"I_SP_T_SPANNSTELLE_3"	M 355.6	BOOL	// M-EINGANG: Spannhydraulik Taster Spannstelle 3
"I_SP_T_SPANNSTELLE_4"	M 355.7	BOOL	// M-EINGANG: Spannhydraulik Taster Spannstelle 4
"O_SP_H_SPANNSTELLE_1"	M 356.0	BOOL	// M-AUSGANG: Spannhydraulik Lampe Spannstelle 1
"O_SP_H_SPANNSTELLE_2"	M 356.1	BOOL	// M-AUSGANG: Spannhydraulik Lampe Spannstelle 2
"O_SP_H_SPANNSTELLE_3"	M 356.2	BOOL	// M-AUSGANG: Spannhydraulik Lampe Spannstelle 3
"O_SP_H_SPANNSTELLE_4"	M 356.3	BOOL	// M-AUSGANG: Spannhydraulik Lampe Spannstelle 4
"O_SP_MPL_ENTKUPPELN"	M 356.4	BOOL	// M-AUSGANG: SpannHydraulik Maschinenplatz entkuppeln
"O_SP_MPL_KUPPELN"	M 356.5	BOOL	// M-AUSGANG: SpannHydraulik Maschinenplatz kuppeln
"O_SP_RPL_AUFL_ENTSPAN"	M 356.6	BOOL	// M-AUSGANG: Ventil Luft für Auflagenkontrolle gelöst am Rüstplatz
"O_SP_RPL_AUFL_SPANNEN"	M 356.7	BOOL	// M-AUSGANG: Ventil Luft für Auflagenkontrolle gespannt am Rüstplatz
"I_AL_ANWAHL_BA1"	M 357.0	BOOL	// M-EINGANG: Freigabe Drehzahl Maximum
"I_AL_ANWAHL_BA2"	M 357.1	BOOL	// M-EINGANG: Freigabe Betriebsart 2
"I_AL_ANWAHL_BA3/4"	M 357.2	BOOL	// M-EINGANG: Freigabe Betriebsart 3/4
"I_PW_MPL_MDK_GEKUPPELT"	M 357.3	BOOL	// M-EINGANG: Medienkupplung Fraes-Drehtisch ausgefahren
"O_SP_RPL_DRUCK_AUS"	M 357.4	BOOL	// M-AUSGANG: H4-29.1 Spanndruck Rüstplatz Aus
"O_SP_RPL_ENTKUPPELN"	M 357.5	BOOL	// M-AUSGANG: SpannHydraulik Rüstplatz entkuppeln
"O_SP_RPL_KUPPELN"	M 357.6	BOOL	// M-AUSGANG: SpannHydraulik Rüstplatz kuppeln
"O_SP_RPL_BLASLUFT"	M 357.7	BOOL	// M-AUSGANG: Ventil Luft für Vorrichtung Abblasen
"O_SP_RPL_FREIGABE"	M 358.0	BOOL	// M-AUSGANG: Freigabe SpannHydraulik Rüstplatz
"O_RPL_TUER_SCHLIESSEN"	M 358.1	BOOL	// M-AUSGANG: Ventil Rüstplatztür schließen
"O_SO_WFK_KLE_KLEMMEN"	M 358.2	BOOL	// M-AUSGANG: Wiegenfräskopf Klemmung klemmen
"O_SO_WFK_KLE_LOESEN"	M 358.3	BOOL	// M-AUSGANG: Wiegenfräskopf Klemmung lösen
"O_SO_WFK_MEDIENK_REINIG"	M 358.4	BOOL	// M-AUSGANG: Wiegenfräskopf Medienkupplung abblasen/reinigen
"O_SO_WFK_PNEUMATIK_EIN"	M 358.5	BOOL	// M-AUSGANG: Wiegenfräskopf Pneumatik Ein
"O_SO_DMS_PNEUMAK_EIN"	M 358.6	BOOL	// M-AUSGANG: Drehmomentstütze Pneumatikversorgung Ein
"O_PW_MPL_MDK_ENTKUPPELN"	M 358.7	BOOL	// M-AUSGANG: Medienkupplung Fraes-Drehtisch einfahren
"I_KA_N_SPI_DURCHFLUSSW"	M 359.0	BOOL	// M-EINGANG: Durchflusswaechter Kuehlkreislauf Hauptantrieb
"I_FD_N_DURCHFL_LAGER"	M 359.1	BOOL	// M-EINGANG: Durchflusswaechter Kuehlkreislauf Lager FD-Tisch
"I_FD_NEG_DURCHFL_STATOR"	M 359.2	BOOL	// M-EINGANG: Durchflusswaechter Kuehlkreislauf Stator FD-Tisch
"I_KA_N_ACHS_DURCHFLUSSW"	M 359.3	BOOL	// M-EINGANG: Durchflusswaechter Kuehlkreislauf Vorschubantriebe
"I_AL_N_FLOW_SWITCH_3"	M 359.4	BOOL	// M-EINGANG:
"I_FD_D_TISCH_GEKLEMMT"	M 359.5	BOOL	// M-EINGANG: Diagnose Klemmung geklemmt
"I_FD_D_TISCH_GELOEST"	M 359.6	BOOL	// M-EINGANG: Diagnose Klemmung geloest
"I_FD_SCH_ZYL_SCHALTER"	M 359.7	BOOL	// M-EINGANG: Zyklenschalter Progressivverteiler
"I_FD_SCH_FUELL_OK"	M 360.0	BOOL	// M-EINGANG: Fuellstand Schmierstoffpumpe Fraes-Drehtisch
"O_WFK_aktiv"	M 360.1	BOOL	// WIKO: Betrieb mit aktivem Wiegenfräßkopf
"I_SP_SPANN_LOES"	M 360.2	BOOL	// M-EINGANG: Wahlschalter Spannhydraulik
"I_SP_AKTIV"	M 360.3	BOOL	// M-EINGANG: Freigabe Sicherheitsventil
"O_KM_FEINSTB_PUMPE"	M 360.4	BOOL	// M-AUSGANG: Foerderpumpe Feinstbereich
"O_FD_SCH_PUMPE_EIN"	M 360.5	BOOL	// M-AUSGANG: Schmierstoffpumpe ein Fraes-Drehtisch
"I_KM_WARN_KSS_TEMP"	M 361.0	BOOL	// M-EINGANG: Kuehlmittel Warnung Temperaturueberwachung
"I_KM_Leckueberw_OK"	M 361.1	BOOL	// M-EINGANG: Ueberwachung Kuehlmittel SFK
"O_PW_MPL_MDK_KUPPELN"	M 361.2	BOOL	// M-AUSGANG: Medienkupplung Fraes-Drehtisch ausfahren
"I_MessDose_BB"	M 361.3	BOOL	// M-EINGANG: Messdose Betriebsbereit
"I_WZ_MIN_SCH_Fuell_OK"	M 361.4	BOOL	// M-EINGANG: Minimalmengenschmierung Fuellstand ok
"I_AL_SCH_M26_Rueckm"	M 361.5	BOOL	// M-EINGANG: Druckueberwachung Schmierung M26 (Drehdurchführung)
"I_AL_SCH_M26_Fuellstand"	M 361.6	BOOL	// M-EINGANG: Schmierung M26 (Drehdurchführung) Füllstand
"I_WS_Grf_offen"	M 363.4	BOOL	// M-EINGANG: STA: Werkstückgreifer geöffnet
"M_FP_Quit_M206"	M 368.0	BOOL	// WIKO: Quittierung M206 Flanke positiv
"M_Quit_M206"	M 368.1	BOOL	// WIKO: Quittierung M206
"I_FD_PW_KLE_geklemmt"	M 368.2	BOOL	// M-EINGANG: Palettenklemmung Fraes-Drehtisch geklemmt
"I_FD_PW_KLE_geloest"	M 368.3	BOOL	// M-EINGANG: Palettenklemmung Fraes-Drehtisch geloest
"I_DM_Ta_Rohteil"	M 368.5	BOOL	// M-EINGANG: MSST: Taste Status Palette Rüstplatz Maschine auf Rohteil setzen
"M_write_siro_db227"	M 368.7	BOOL	// TDS: BALLUFF Ablöschen der Daten im DB227 beim Entladen
"I_DM_Ta Y-Achse plus"	M 370.0	BOOL	// M-EINGANG: MSST: Taste Y-Achse plus
"I_DM_Ta 4-Achse rechts"	M 370.1	BOOL	// M-EINGANG: MSST: Taste 4-Achse rechts
"I_DM_Ta Eilgang"	M 370.2	BOOL	// M-EINGANG: MSST: Taste Eilgang_T 29
"I_DM_Ta_5/6-Achse minus"	M 370.3	BOOL	// M-EINGANG: MSST: Taste 5/6 Achse minus_T 48
"I_DM_Ta_5/6-Achse plus"	M 370.4	BOOL	// M-EINGANG: MSST: Taste 5/6 Achse plus_T 48
"I_DM_Ta X-Achse minus"	M 370.5	BOOL	// M-EINGANG: MSST: Taste X-Achse minus_T 30
"I_DM_Ta X-Achse plus"	M 370.6	BOOL	// M-EINGANG: MSST: Taste X-Achse plus_T 28
"I_DM_Ta Z-Achse minus"	M 370.7	BOOL	// M-EINGANG: MSST: Taste Z-Achse minus_T 39
"I_DM_Ta Z-Achse plus"	M 371.0	BOOL	// M-EINGANG: MSST: Taste Z-Achse plus
"I_DM_Ta 4-Achse links"	M 371.1	BOOL	// M-EINGANG: MSST: Taste 4-Achse links_T 40
"I_DM_Ta Y-Achse minus"	M 371.2	BOOL	// M-EINGANG: MSST: Taste Y-Achse minus_T 38
"I_DM_Ta Spindel rechts"	M 371.3	BOOL	// M-EINGANG: MSST: Taste Spindel links -_T 8
"I_DM_Ta_Spindel links"	M 371.4	BOOL	// M-EINGANG: MSST: Taste Spindel rechts_T 10
"I_DM_Ta_Spindel HALT"	M 371.5	BOOL	// M-EINGANG: MSST: Taste Spindel Halt_T 9
"I_DM_Ta_Spindel_over100"	M 371.6	BOOL	// M-EINGANG: MSST: Taste Spindeloverride 100%
"I_DM_Ta_SpiOVR_erhoehen"	M 371.7	BOOL	// M-EINGANG: MSST: Taste Spindeloverride erhöhen
"I_DM_Ta_SpiOVR_reduz"	M 372.0	BOOL	// M-EINGANG: MSST: Taste Spindeloverride reduzieren
"I_DM_Ta_BHG"	M 372.1	BOOL	// M-EINGANG: MSST: Taste Bedienhandgerät
"I_DM_Ta_KMTL"	M 372.2	BOOL	// M-EINGANG: MSST: Taste Kühlmittel
"I_DM_Ta_IKZ"	M 372.3	BOOL	// M-EINGANG: MSST: Taste Innere Kühlmittel
"O_WK_NOTACHSBETRIEB"	M 373.0	BOOL	// M-AUSGANG: KometU-Achse:Notachsbetrieb
"o_uc2e1"	M 373.1	BOOL	// M-AUSGANG: KometU-Achse:Reserve PosCode 2e1
"o_uc2e2"	M 373.2	BOOL	// M-AUSGANG: KometU-Achse:Reserve PosCode 2e2
"o_uc2e3"	M 373.3	BOOL	// M-AUSGANG: KometU-Achse:Reserve PosCode 2e3
"O_WK_POSITIONIEREN"	M 373.4	BOOL	// M-AUSGANG: KometU-Achse:Reserve PosKommando
"O_WK_PARKEN"	M 373.5	BOOL	// M-AUSGANG: KometU-Achse:Reserve Parkkommando
"O_WK_ACHSBETRIEB"	M 373.6	BOOL	// M-AUSGANG: KometU-Achse:Kommando Achsbetrieb
"O_WK_QUIT_ALARM"	M 373.7	BOOL	// M-AUSGANG: KometU-Achse:Störung quittieren
"I_WK_ALARMCODE_BIT_0"	M 374.0	BOOL	// M-EINGANG: KometU-Achse:Alarmcode Bit 2e0
"I_WK_ALARMCODE_BIT_1"	M 374.1	BOOL	// M-EINGANG: KometU-Achse:Alarmcode Bit 2e1
"I_WK_ALARMCODE_BIT_2"	M 374.2	BOOL	// M-EINGANG: KometU-Achse:Alarmcode Bit 2e2
"I_WK_ALARMCODE_BIT_3"	M 374.3	BOOL	// M-EINGANG: KometU-Achse:Alarmcode Bit 2e3
"I_WK_QUIT_KOMMANDO"	M 374.4	BOOL	// M-EINGANG: KometU-Achse:Quit bei PtP, Reserve
"I_WK_NEG_ALARM"	M 374.5	BOOL	// M-EINGANG: KometU-Achse:Alarm, L-aktiv
"I_WK_NEG_WZ_AKTIV"	M 374.6	BOOL	// M-EINGANG: KometU-Achse:Werkzeug beschäftigt, L-aktiv
"I_WK_WZ_BTB"	M 374.7	BOOL	// M-EINGANG: KometU-Achse:System bereit
"I_WK_REF"	M 375.0	BOOL	// M-EINGANG: KometU-Achse:RefNocken
"I_WK_BTB"	M 375.1	BOOL	// M-EINGANG: KometU-Achse:Achse bereit
"I_WK_ENDSCHALTER_PLUS"	M 375.2	BOOL	// M-EINGANG: KometU-Achse:Vorendschalter positiv
"I_WK_ENDSCHALTER_MINUS"	M 375.3	BOOL	// M-EINGANG: KometU-Achse:Vorendschalter negativ
"m375.4"	M 375.4	BOOL	// M-EINGANG: KometU-Achse: Reserve
"m375.5"	M 375.5	BOOL	// M-EINGANG: KometU-Achse: Reserve
"m375.6"	M 375.6	BOOL	// M-EINGANG: KometU-Achse: Reserve
"m375.7"	M 375.7	BOOL	// M-EINGANG: KometU-Achse: Reserve
"m_WzwSpUAx"	M 376.0	BOOL	// KOMET U-ACHSE: Werkzeugwechsel sperren, Komet-U-Achse in Spindel.& aktiv
"m_UiSpi"	M 376.1	BOOL	// KOMET U-ACHSE: Komet-U-Achse Werkzeug in Spindel
"m_UNotBt"	M 376.2	BOOL	// KOMET U-ACHSE: Notbetrieb von Bediener gewählt
"m_LSpUAx"	M 376.3	BOOL	// KOMET U-ACHSE: Einlesesperre durch Komet U-Achse
"M_MAG_Umk_Korrektur_bei+"	M 376.4	BOOL	// MAG: Korrektur Umkehrspiel: Aktivierung bei Plusfahrt
"M_MAG_Umk_Korrektur_bei-"	M 376.5	BOOL	// MAG: Korrektur Umkehrspiel: Aktivierung bei Minusfahrt
"M_MAG_Umk_+-1_plz_ang"	M 376.6	BOOL	// MAG: Umkehrspiel: +/- 1 Platz fahren angewählt
"M_MAG_Umk_rueck_auf_plz"	M 376.7	BOOL	// MAG :Korrektur Umkehrspiel: Rückfahrt auf vorgegebenen Mag-Platz angewählt
"M_Bearb_Ende"	M 377.0	BOOL	// SINRPC: Bearbeitungsprogramm Ende
"M_Drehzahl_Sperre"	M 377.1	BOOL	// SPINDEL: Drehzahlsperre
"M_MAG_Umk_reset_korr_fp"	M 377.2	BOOL	// MAG: Korrektur Umkehrspiel: Reset Flanke Positiv
"M_MAG_Umk_kuerzesterWeg+"	M 377.3	BOOL	// MAG: Korrektur Umkehrspiel: kürzester Weg Magazinachse ins Plus
"M_MAG_Umk_kuerzesterWeg-"	M 377.4	BOOL	// MAG: Korrektur Umkehrspiel: kürzester Weg Magazinachse ins Minus
"M_MAG_Teller_Taste_dreh"	M 377.6	BOOL	// MAG: Tellermagazin Anforderung drehen über Taste
"Mx_Maschine_min_1mal_ein"	M 377.7	BOOL	// SINRPC: Maschine min einmal ein
"O_TM_TOOL_SPIPOS_LOCK"	M 378.0	BOOL	// Verriegelungszylinder ausfahren (Werkzeug verriegeln)
"I_TM_TOOL_SPIPOS_UNLKD"	M 378.1	BOOL	// eingefahren (Werkzeug entriegelt)
"I_TM_TOOL_SPIPOS_LOCKED"	M 378.2	BOOL	// ausgefahren (Werkzeug entriegelt)
"I_TM_TST_OCC"	M 378.3	BOOL	// M-EINGANG: Uebergabeplatz belegt vertikale Kette ohne TPU
"M_RS_HUBACHSE_E0_UNTEN"	M 379.0	BOOL	// PALETTENSPEICHER: Hubachse in Ebene 0 unten
"M_RS_HUBACHSE_E0_OBEN"	M 379.1	BOOL	// PALETTENSPEICHER: Hubachse in Ebene 0 oben
"M_RS_HUBACHSE_E1_UNTEN"	M 379.2	BOOL	// PALETTENSPEICHER: Hubachse in Ebene 1 unten
"M_RS_HUBACHSE_E1_OBEN"	M 379.3	BOOL	// PALETTENSPEICHER: Hubachse in Ebene 1 oben
"O_SST_SC_CL_PO_1_STATE"	M 379.4	BOOL	// MA H4-93.2 Status Auflagenkontrolle Spannstelle 1 (Meldeleuchte)
"O_SST_SC_CL_PO_2_STATE"	M 379.5	BOOL	// MA H4-93.4 Status Auflagenkontrolle Spannstelle 2 (Meldeleuchte)
"O_SST_FLUSH_ON_H"	M 379.7	BOOL	// MA B2-87.6 Ruestplatz Spuelung aktiv (Meldeleuchte)
"O_SP_HYD_RPL_LOESEDR_OK"	M 382.0	BOOL	// M-AUSGANG: Spannvorrichtung Loesedruck vorhanden
"O_SP_HYD_RPL_SPANNDR_OK"	M 382.1	BOOL	// M-AUSGANG: Spannvorrichtung Spanndruck vorhanden
"I_PW_HUB_POS1"	M 382.2	BOOL	// M-EINGANG: Palettenwechsler Hub Position 1
"I_PW_HUB_POS2"	M 382.3	BOOL	// M-EINGANG: Palettenwechsler Hub Position 2
"I_PW_HUB_POS3"	M 382.4	BOOL	// M-EINGANG: Palettenwechsler Hub Position 3
"I_SP_HYD_EIN"	M 382.5	BOOL	// M-EINGANG: Bereichsschalter Spannhydraulik Ein
"I_SP_HYD_FUEL_OK"	M 382.6	BOOL	// M-EINGANG: Spannhydraulik Ueberwachung Fuellstand
"I_SP_HYD_NEG_STOERUNG"	M 382.7	BOOL	// M-EINGANG: Spannhydraulik Motorschutzschalter ok
"I_SP_HYD_RPL_LOESEN"	M 383.0	BOOL	// M-EINGANG: Fußschalter Spannhydraulik entspannen (lösen)
"I_SP_HYD_RPL_SPANNEN"	M 383.1	BOOL	// M-EINGANG: Fußschalter Spannhydraulik spannen
"I_SP_HYD_TEMP_OK"	M 383.2	BOOL	// M-EINGANG: Spannhydraulik Temperatur ok
"M_FP_PW_Step_Forward"	M 383.3	BOOL	// PW: Schritt Vorwärts Flanke positiv
"M_FP_PW_Step_Backward"	M 383.4	BOOL	// PW: Schritt Rückwärts Flanke positiv
"M_FN_PW_Step_Forward"	M 383.5	BOOL	// PW: Schritt Vorwärts Flanke negativ
"M_FN_PW_Step_Backward"	M 383.6	BOOL	// PW: Schritt Rückwärts Flanke negativ
"O_SP_SPANNVORR_RV_EIN"	M 383.7	BOOL	// M-AUSGANG: Rückschlagventil Entspann-Leitung RPL öffnen
"Mx_APC_Disable_H67"	M 384.0	BOOL
"Mx_Pal_Fertigteil_H67"	M 384.1	BOOL
"Mx_Pal_Defekt_H67"	M 384.2	BOOL
"O_WK_KOPF_ANGEBAUT"	M 384.4	BOOL	// M-AUSGANG: U-Achse Werkzeug angebaut
"O_WK_REG_FREIGABE"	M 384.5	BOOL	// M-AUSGANG: U-Achse Reglerfreigabe
"O_SST_FIXT_CL_PO_1_CLE"	M 384.6	BOOL	// MA H4-94.2 Auflagenkontrolle Luft für Reinigung (hoher ALK-Druck)
"O_SST_SC_SENS_ACT"	M 384.7	BOOL	// MA H4-94.4 Auflagenkontrolle Luft für Messung (niedriger ALK-Druck)
"m_mag_handfunktion_-"	M 385.0	BOOL	// MAG: Handfunktion Magazinachse ins Minus drehen
"m_mag_handfunktion_+"	M 385.1	BOOL	// MAG: Handfunktion Magazinachse ins Plus drehen
"m_mag_positioniert_fp"	M 385.2	BOOL	// MAG: Handfunktion Magazinachse positioniert Flanke positiv
"M_Tast_Man_WZSp"	M 386.0	BOOL	// WZ-SPANNER:Werkzeugspanner manuell lösen
"MX_Temp_Vorw"	M 386.1	BOOL	// KM: KSA3 Vorwarnung Temporär
"M_Motor_Aus"	M 386.2	BOOL	// KM: KSA3 Motor Aus Temporär
"I_SO_WFK_ANGEDOCKT"	M 386.3	BOOL	// M-EINGANG: Wiegenfräskopf angedockt / Klemmposition erreicht
"I_SO_WFK_KLE_GEKLEMMT"	M 386.4	BOOL	// M-EINGANG: Wiegenfräskopf Klemmung geklemmt
"I_SO_WFK_KLE_GELOEST"	M 386.5	BOOL	// M-EINGANG: Wiegenfräskopf Klemmung gelöst
"I_SO_DMS_UEBERWACH_OEL"	M 386.6	BOOL	// M-EINGANG: Drehmomentstütze Ölstandsüberwachung Niveau
"I_AL_NETZAUSF_UEBERW"	M 386.7	BOOL	// ME A0-82.4 Spannungsüberwachung Netz nicht in Ordnung
"I_SP_HYD_RPL_AUS"	M 387.0	BOOL	// M-EINGANG: Ruestplatz Ventil Drucklos
"I_HYD_NEG_FILTER_RPL"	M 387.1	BOOL	// M-EINGANG: Spannhydraulik Filterverschmutzung Ruestplatz
"I_HYD_NEG_FILTER_MPL"	M 387.2	BOOL	// M-EINGANG: Spannhydraulik Filterverschmutzung Maschinenplatz
"I_ACHS_PNOZ_FRG"	M 387.3	BOOL	// M-EINGANG: Freigabe Achsen Sicherheitsschaltgeraet
"O_SP_RPL_GESPANNT"	M 387.4	BOOL	// M-AUSGANG: Spannhydraulik Ruestplatz gespannt
"O_SP_RPL_DRUCKLOS"	M 387.5	BOOL	// M-AUSGANG: Ruestplatz Ventil Drucklos
"O_SP_MPL_DRU_OK"	M 387.6	BOOL	// M-AUSGANG: Spannvorrichtung Maschine gespannt
"O_SP_RPL_SPANNEN"	M 387.7	BOOL	// Spannhydraulik Ruestplatz spannen
"O_SP_MASCHINE_ENTLADEN"	M 388.0	BOOL	// M-AUSGANG: H4-07.6 Rueckmeldung Maschine Entladen
"O_SP_SCH_EIN"	M 388.1	BOOL	// M-AUSGANG: H4-05.2 Schmierstoffpumpe Spannfutter Spannvorrichtung
"M_Vollwechsel_beendet"	M 388.2	BOOL
"M_FP_Vollwechsel_beendet"	M 388.3	BOOL
"I_AL_WARNMELD_PWR_SAG"	M 389.0	BOOL	// Spannungsüberwachung Netz
"I_SP_MASCHINE_ENTLADEN"	M 389.1	BOOL	// Maschine Entladen
"I_SP_SCH_DRUCK_OK"	M 389.2	BOOL	// Druckueberwachung Schmierung Spannfutter
"I_SP_SCH_FUELLSTAND_OK"	M 389.3	BOOL	// M-EINGANG: H4-05.5 Fuellstand Schmierung Spannfutter
"M_FP_WARN_PWR_SAG"	M 389.4	BOOL	// Positive Flanke Spannungsüberwachung Netz
"M_FP_Warnmeldung_Netz"	M 389.5	BOOL	// Impuls Spannungsüberwachung Netz
"MX_BHG_aktiv"	M 390.0	BOOL	// BHG-MPI: aktiv
"MX_FP_BHG_aktiv"	M 390.1	BOOL	// BHG-MPI: aktiv Flanke positiv
"MX_FN_BHG_aktiv"	M 390.2	BOOL	// BHG-MPI: aktiv Flanke negativ
"MX_BHG_Reset"	M 390.3	BOOL	// BHG-MPI: Reset
"MX_BHG_Anf_JOG"	M 390.4	BOOL	// BHG-MPI: Anforderung JOG
"MX_BHG_Anf_Single"	M 390.5	BOOL	// BHG-MPI: Anforderung Single Block
"MX_BHG_KM1_EinAus"	M 390.6	BOOL	// BHG-MPI: Taste Kühlmittel Ein / Aus
"MX_BHG_Handrad_aktiv"	M 390.7	BOOL	// BHG-MPI: Handrad aktiv
"MX_BHG_Taste_plus"	M 391.0	BOOL	// BHG-MPI: Taste Plus
"MX_BHG_Taste_minus"	M 391.1	BOOL	// BHG-MPI: Taste Minus
"MX_BHG_X_Vorwahl"	M 391.2	BOOL	// BHG-MPI: Vorwahl X-Achse
"MX_BHG_Y_Vorwahl"	M 391.3	BOOL	// BHG-MPI: Vorwahl Y-Achse
"MX_BHG_Z_Vorwahl"	M 391.4	BOOL	// BHG-MPI: Vorwahl Z-Achse
"MX_BHG_C_Vorwahl"	M 391.5	BOOL	// BHG-MPI: Vorwahl C-Achse
"MX_BHG_5/6_Vorwahl"	M 391.6	BOOL	// BHG-MPI: Vorwahl 5te / 6te Achse
"MX_BHG_Taste_INC1000"	M 391.7	BOOL	// BHG-MPI: Taste INC1000
"MX_BHG_Anf_INC_100"	M 392.0	BOOL	// BHG-MPI: Anforderung INC100
"MX_BHG_Anf_INC_10"	M 392.1	BOOL	// BHG-MPI: Anforderung INC10
"MX_BHG_Anf_INC_1"	M 392.2	BOOL	// BHG-MPI: Anforderung INC1
"MX_BHG_Anf_VorschHalt"	M 392.3	BOOL	// BHG-MPI: Anforderung Vorschub Halt
"MX_BHG_Anf_VorschStart"	M 392.4	BOOL	// BHG-MPI: Anforderung Vorschub Start
"MX_BHG_Anf_SpindelStart"	M 392.5	BOOL	// BHG-MPI: Anforderung Spindel Start
"MX_BHG_Anf_NC-Start"	M 392.6	BOOL	// BHG-MPI: Anforderung NC-Start
"MX_BHG_Anf_NC-Stop"	M 392.7	BOOL	// BHG-MPI: Anforderung NC-Stop
"MX_BHG_Taste_Eilgang"	M 393.0	BOOL	// BHG-MPI: Taste Eilgang
"MX_BHG_Anf_INC_1000"	M 393.1	BOOL	// BHG-MPI: Anforderung INC1000
"MX_WKS_MKS_Aend"	M 393.2	BOOL	// BHG-MPI: WKS / MKS Änderung
"MX_AX4_InPos_Fein"	M 393.3	BOOL	// BHG-MPI: Achse 4 Position erreicht mit Genauhalt fein
"MX_AX5_InPos_Fein"	M 393.4	BOOL	// BHG-MPI: Achse 5 Position erreicht mit Genauhalt fein
"MX_NC_Datueb_aktiv"	M 393.5	BOOL	// BHG-MPI: NC Datenübertragung aktiv
"MX_RD_akt_Pos_MKS"	M 393.6	BOOL	// BHG-MPI: Aktuelle Position MKS
"M_Error_WR_FC13"	M 393.7	BOOL	// BHG-MPI: Fehler Displaycontrol
"MX_RD_akt_Pos_WKS"	M 394.0	BOOL	// BHG-MPI: Aktuelle Position MKS
"M_Initialisier_Auftraege"	M 394.1	BOOL	// WIKO: Aufträge initialisieren
"I_KM_DURCHFLUSS_HD_OK"	M 394.2	BOOL	// M-EINGANG: ME C1-13.4 Durchflusswaechter Kuehlmittel 2 (M7)
"I_KM_M7_DFW_LTG_OK"	M 394.3	BOOL	// M-EINGANG: ME C1-13.7 Durchflusswaechter Leitungsueberwachung (M7)
"M_Restweg_aktiv"	M 394.4	BOOL
"M_Error_Restweg_lesen"	M 394.5	BOOL
"M_NDR_Restweg_lesen"	M 394.6	BOOL
"M_Req_Restweg_lesen"	M 394.7	BOOL
"O_SO_EXH_ON1"	M 397.0	BOOL	// Leistungssteuerung Absauganlage
"O_MT_KALIBRIER_REINIGEN"	M 397.1	BOOL	// Kalibrier Vorrichtung Messtaster abblasen
"I_KM_WARTUNG"	M 397.2	BOOL	// Filterverschmutzung Feinstbereich Warnung
"FP_SS_ROB_OFF"	M 397.3	BOOL	// Flankenmerker positiv Schlüsselschalter Robbi Aus
"FP_SS_RO"	M 397.4	BOOL	// Flankenmerker positiv Schlüsselschalter Robbi Aus
"Mx_PAldata_FASTEMS"	M 400.0	BOOL
"M_FP_Achse4_Spindel"	M 400.1	BOOL
"M_IMP_Achse4_Spindel"	M 400.2	BOOL
"M_FN_Achse4_Spindel"	M 400.3	BOOL
"M_IMP_Achse4_Achse"	M 400.4	BOOL
"M_Axpos_lesen_ready"	M 400.5	BOOL	// UT: Istwert Teil 1 gelesen
"M_184.0"	M 400.6	BOOL	// UT: NC-Datenübertragung aktiv
"M_185.6"	M 400.7	BOOL	// UT: lesen Istwert alle Achsen
"M_Axpos_read_error"	M 401.0	BOOL	// UT: Fehler Istwert lesen
"M_Req_Lesen_Ax9"	M 401.1	BOOL
"M_Error_Lesen_Ax9"	M 401.2	BOOL
"M_RDY_Lesen_Ax9"	M 401.3	BOOL
"MX_Error_RD_IstPos15"	M 401.4	BOOL
"Error_FB_SIEM_GET"	M 401.5	BOOL	// Error-Meldung Baustein FB_SIEM_GET
"NDR_FB_SIEM_GET"	M 401.6	BOOL	// NDR-Meldung Baustein FB_SIEM_GET
"MX_NDR_RD_IstPos15"	M 401.7	BOOL
"M_all_axis_pos_contr_act"	M 402.0	BOOL	// Alle aktiven Achsen befinden sich in Lageregelung
"M_PV_akt_Prg_lesen"	M 404.0	BOOL	// lesen Programmnr. aktives laufendes Programm
"M_FP_BlockSearch"	M 404.1	BOOL	// FP Satzsuchlauf aktiv
"M_M60_angewaehlt"	M 404.2	BOOL
"M_PrgLesenNCbeendet"	M 404.3	BOOL
"M_PrgLesenNC_wiederh"	M 404.4	BOOL	// Programmnummer NC lesen wiederholen bei Fehler
"M_PrgLesenNC_Fehler"	M 404.5	BOOL	// Programmnummer NC lesen Fehler gespeichert
"M_Error_Lesen_Ax16"	M 404.6	BOOL
"M_RDY_Lesen_Ax16"	M 404.7	BOOL
"M_RESET_AX16_SWN_OK"	M 405.0	BOOL
"Mx_FP_aus_Loch"	M 405.1	BOOL	// Werkzeugachse Rettung Flanke positiv
"Mx_FN_Taste"	M 405.2	BOOL	// Werkzeugachse Rettung Flanke negativ
"Mx_FN_Taste_WZ_Achse_RET"	M 405.3	BOOL	// Werkzeugachse Rettung Impuls negativ
"M_AX16_SW_NOCKEN_OK"	M 405.4	BOOL
"M_ANF_Lesen_AX16_CAM"	M 405.5	BOOL
"M_Error_Lesen_Ax16_CAM"	M 405.6	BOOL
"M_RDY_Lesen_Ax16_CAM"	M 405.7	BOOL
"M_Prog_load_unload_ok"	M 406.1	BOOL	// NC-Programm laden / entladen ok
"M_Prog_unloaded"	M 406.5	BOOL	// NC-Programm entladen
"M_Prog_loaded"	M 406.6	BOOL	// NC-Programm geladen
"I_TM_PLACE_OCCUPIED"	M 411.0	BOOL	// M-EINGANG: Magazinplatz belegt
"I_KM_DRUCK0_M7_ENABLE"	M 413.0	BOOL
"M_FN_Komet_vorhanden"	M 413.1	BOOL	// HM neg.Flanke Komet vorhanden
"Mx_SPH_DRUCK0_GESAMT_RPL"	M 413.2	BOOL	// Maschinenplatz: alle konfigurierten Spannstellen haben "Druck 0"
"Mx_SPH_DRUCK0_GESAMT_MPL"	M 413.3	BOOL	// Maschinenplatz: alle konfigurierten Spannstellen haben "Druck 0"
"I_PW_SCH_FUELLSTAND"	M 413.5	BOOL	// M-EINGANG: Schmierung Palettenwechsler Überwachung Füllstand
"I_PW_SCH_RUECKMELDUNG"	M 413.6	BOOL	// M-EINGANG: Schmierung Palettenwechsler Drucküberwachung
"O_PW_SCH_PUMPE_EIN"	M 413.7	BOOL	// M-AUSGANG: Schmierung Palettenwechsler
"I_PW_HUB_2_MITTE"	M 414.0	BOOL	// M-EINGANG: Palettenwechsler Position vor Mitte
"I_PW_HUB_2_UNTEN"	M 414.1	BOOL	// M-EINGANG: Palettenwechsler Position vor unten
"O_PW_HUB_2_HEBEN"	M 414.2	BOOL	// M-AUSGANG: Palettenwechsler Hubeinheit nach oben schnell
"O_PW_HUB_2_SENKEN"	M 414.3	BOOL	// M-AUSGANG: Palettenwechsler Hubeinheit nach unten schnell
"M_FN_KNOLL_ERROR"	M 414.4	BOOL	// KM: KNOLL Fehler Flanke negativ
"M_KNOLL_ERROR"	M 414.5	BOOL	// KM: KNOLL Fehler steht an
"M_PS_RPL_BLASLUFT_PARALL"	M 414.6	BOOL	// PALETTENSPEICHER: Blasluft Medienkupplung einschalten
"Error_FB_SIEM_GET_WZDat"	M 421.0	BOOL	// WZV: Error Greiferdaten lesen 2
"NDR_FB_SIEM_GET_WZDat"	M 421.1	BOOL	// WZV: Greiferdaten lesen fertig 2
"Req_FB_SIEM_GET_WZDat"	M 421.2	BOOL	// WZV: Request Greiferdaten lesen 2
"M_Taste_TLOAD_TOOL_LOCK"	M 421.3	BOOL
"M_FP_Zustimmtaste"	M 421.4	BOOL
"M_IM_Zustimmtaste"	M 421.5	BOOL
"M_Sperre_entr_Ladest"	M 421.6	BOOL
"M_FP_WM_Tuere_zu"	M 421.7	BOOL
"M_FP_SPH_FD_entspannen"	M 426.0	BOOL	// Impuls Spannhydraulik FD entspannen
"M_FP_Rein_Ende"	M 426.6	BOOL
"M_FN_Rett_Rein"	M 426.7	BOOL
"I_RPT_Taste_Pal_drehen"	M 427.0	BOOL	// ME xx-xx.x Taste Palette am RPL über NC-Achse drehen
"m_Req_RPAchse_drehen"	M 427.1	BOOL	// Anforderung Palette am RPL über NC-Achse drehen
"M_FP_WZ_Vorbereitet"	M 430.0	BOOL	// WZV: Quittung Bereitstellen fertig Flanke positiv
"M_FP_Reset_WZVorbereitet"	M 430.1	BOOL	// WZV: Reset Bereitstellen fertig Flanke positiv
"O_SF_Schnecke2_Maschine"	M 430.2	BOOL	// M-AUSGANG: Spaenefoerderer Schneckenantrieb 2 ein
"O_SF_Schnecke_Maschine"	M 430.3	BOOL	// M-AUSGANG: Spaenefoerderer Schneckenantrieb ein
"M_A4_loes_aktiv"	M 430.4	BOOL	// AX: Achse 4 lösen aktiv
"M_WZGr1_belegt"	M 430.5	BOOL	// WZW: Greifer 1 hat ein Werkzeug
"M_WZGr2_belegt"	M 430.6	BOOL	// WZW: Greifer 2 hat ein Werkzeug
"M_Req_GRF2_Mag"	M 430.7	BOOL	// WZW: Anforderung Greifer 2 zum Magazin
"M_FN_SPI_re.li."	M 431.0	BOOL	// MSST: Taste Spindel links / rechts Flanke negativ
"O_AL_5ACHS_KLE_LOESEN"	M 431.1	BOOL	// Klemmung loesen NC-Teilapparat
"M_WZWV_UMSPEICHERN"	M 431.2	BOOL	// WZWV: Gr2-->TPU Gr1-->Spdl / Gr1-->TPU Gr2-->Spdl Umspeichern aktivieren
"M_FP_SOKO_ERROR1"	M 431.3	BOOL	// SONDERKONSTRUKTION: SOKO Fehler 1 Flanke positiv
"M_FP_SOKO_ERROR2"	M 431.4	BOOL	// SONDERKONSTRUKTION: SOKO Fehler 2 Flanke positiv
"M_FP_KNOLL_ERROR1"	M 431.5	BOOL	// KM: KNOLL Fehler 1 Flanke positiv
"M_FP_KNOLL_ERROR2"	M 431.6	BOOL	// KM: KNOLL Fehler 2 Flanke positiv
"M_M_FKT_SPANNER_ZU_FP"	M 431.7	BOOL	// WZWV: M-Funktion Werkzeugspanner schliessen Flanke positiv
"O_AL_KABINE_ENTRIEGELN"	M 432.0	BOOL	// M-AUSGANG: Magnetverriegelung Kabinentüre entriegeln
"O_AL_PLC_BTB"	M 432.1	BOOL	// M-AUSGANG: Maschine 'Ein'  (CNC PLC Betriebsbereit)
"O_AL_Manual_Betrieb"	M 432.2	BOOL	// M-AUSGANG: Handbetrieb (Manual)
"O_Umsch_Zustimm_HR"	M 432.3	BOOL	// M-AUSGANG: Handkommandostation angewählt /Umschaltung Zustimmtasten
"O_AL_SCH_Pumpe_ein"	M 432.4	BOOL	// M-AUSGANG: Schmierung Maschine 'Ein'
"O_AL_Tempkomp_DSR"	M 432.5	BOOL	// M-AUSGANG: Temperaturkompensation rücksetzen Synchronisation Temperaturdaten
"O_AL_Tempkomp_CTS"	M 432.6	BOOL	// M-AUSGANG: Temperaturkompensation   Temperaturdaten auslesen
"M_SOKO_ERROR"	M 432.7	BOOL	// SONDERKONSTRUKTION: SOKO Fehler
"O_SK_1_Stufe_Getriebe"	M 433.0	BOOL	// M-AUSGANG: Drehzahlschaltung Hauptantrieb mit Getriebe    Drehzahl kleiner
"O_SK_2_Stufe_Getriebe"	M 433.1	BOOL	// M-AUSGANG: Drehzahlschaltung Hauptantrieb mit Getriebe    Drehzahl größer
"O_AL_Druckluft_ein"	M 433.2	BOOL	// M-AUSGANG: Pneumatik 'Ein'
"O_AL_Hydraulik_Ein"	M 433.3	BOOL	// M-AUSGANG: Hydraulik 'Ein'
"O_AL_WZ_Spanner_Loesen"	M 433.4	BOOL	// M-AUSGANG: Werkzeugspanner lösen (Autobetr)/Anwahl lösen (Handbetr)
"O_4_Klem_Bremse_Auf"	M 433.5	BOOL	// M-AUSGANG: 4.Achse Klemmung lösen
"O_5_Klem_Bremse_Auf"	M 433.6	BOOL	// M-AUSGANG: 5./11. Achse Klemmung lösen
"O_AL_Start_Sig_Renishaw"	M 433.7	BOOL	// M-AUSGANG: Messtasterfreigabe
"O_WZKegel_Blasluft"	M 434.0	BOOL	// M-AUSGANG: Messtaster Messstelle reinigen (M29) und  Werkzeugkegel ausblasen
"O_KM_M8_Ein"	M 434.1	BOOL	// M-AUSGANG: Pumpe Kühlmittel 1 'Ein' (M8)
"O_KM_M7_Ein"	M 434.2	BOOL	// M-AUSGANG: Pumpe Kühlmittel 2 'Ein' (M7)
"M_M8_Sperre_Wiko"	M 434.3	BOOL
"O_SFK_Hori_schwenken"	M 434.4	BOOL	// SCHWENKFRÄSKOPF: schwenken waagrecht (M53)
"M_M7_aktivieren_Wiko"	M 434.5	BOOL
"O_SFK_Klemmung_zu"	M 434.6	BOOL	// SCHWENKFRÄSKOPF: Klemmung klemmen
"O_SFK_Klemmung_Auf"	M 434.7	BOOL	// SCHWENKFRÄSKOPF: Klemmung lösen
"O_SPI_SCH_OEL"	M 435.0	BOOL	// M-AUSGANG: Schmierung Hauptantrieb 24.000 U/min
"O_SPI_SCH_LUFT"	M 435.1	BOOL	// M-AUSGANG: Schwenkfräskopf Druckluft Schmierung 'Ein'
"M_FR_PW_HA_SYST"	M 435.2	BOOL	// Freigabe Palettenwechsel vom Handlingsystem
"M_FN_Be_Entladen"	M 435.3	BOOL	// Abfallende Flanke: Be- Entladen aktiv
"O_Programm_Ende"	M 435.4	BOOL	// MA: Zusatzfunktion Programm Ende (M30)
"O_CNC_Fehlermeldung"	M 435.5	BOOL	// MA: Zusatzfunktion NC-Fehlermeldung steht an
"O_Funktion_M190"	M 435.6	BOOL	// M-AUSGANG: Zusatzfunktion M190
"O_PC_PAL_CAR_DOWN"	M 435.7	BOOL	// M-AUSGANG: Takttisch Palettenträger senken
"O_WM_MAG_Rechtslauf"	M 436.0	BOOL	// M-AUSGANG: Werkzeugmagazin Rechtslauf
"O_WM_MAG_Linkslauf"	M 436.1	BOOL	// M-AUSGANG: Werkzeugmagazin Linkslauf
"O_KA_STOERMELDUNG1"	M 436.2	BOOL	// M-AUSGANG: Kuehlaggregat Störmeldung Prioritaet 1
"O_PW_SPANNDRUCK_HYD_AUS"	M 436.3	BOOL	// M-AUSGANG: MA H4-03.7 Spannvorrichtung Verriegelung Palettenwechsler
"O_WZ_DATENSICHERUNG"	M 436.7	BOOL	// M-AUSGANG: Anstoss zur Datensicherung der Werkzeugdaten
"O_PW_PAL_AUF_RP_SPANNEN"	M 437.0	BOOL	// M-AUSGANG: Palette auf Rüstplatz spannen
"O_PW_PAL_AUF_RP_LOESEN"	M 437.1	BOOL	// M-AUSGANG: Palette auf Rüstplatz lösen
"O_PW_ANDOCK_SENKEN"	M 437.2	BOOL	// M-AUSGANG: Palettenwechsler Rüstplatz Andockstation senken
"O_PW_ANDOCK_HEBEN"	M 437.3	BOOL	// M-AUSGANG: Palettenwechsler Rüstplatz Andockstation heben
"O_PW_FREIGABE"	M 437.4	BOOL	// M-AUSGANG: Anforderung Freigabe Palettenwechsel
"O_WZB_Abblasen"	M 437.5	BOOL	// M-AUSGANG: Werkzeugbruchkontrolle abblasen
"O_AL_4_BA_Selbsthaltung"	M 437.7	BOOL	// M-AUSGANG: Energiefreigabe 4.Betriebsart
"O_WZB_Messung_Start"	M 438.0	BOOL	// M-AUSGANG: Werkzeugbruchüberwachung Freigabe
"O_Fenster_WZ_Mag_zu"	M 438.1	BOOL	// M-AUSGANG: Magnetverriegelung Fenster Werkzeugbestückung
"O_WM_Beladung_entr_auf"	M 438.2	BOOL	// M-AUSGANG: Freigabe Magnetverriegelung Fenster Werkzeugbestückung
"O_PW_KLE_loesen"	M 438.3	BOOL	// M-AUSGANG: Palette auf Tisch lösen
"O_PW_KLE_klemmen"	M 438.4	BOOL	// M-AUSGANG: Palette auf Tisch spannen
"O_PW_Hub_senken"	M 438.5	BOOL	// M-AUSGANG: Palettenwechsler nach unten
"O_PW_Hub_heben"	M 438.6	BOOL	// M-AUSGANG: Palettenwechsler nach oben
"O_PW_0_Grad_Drehen"	M 438.7	BOOL	// M-AUSGANG: Palettenwechsler schwenken 0 Grad Position
"O_PW_180_Grad_Drehen"	M 439.0	BOOL	// M-AUSGANG: Palettenwechsler schwenken 180 Grad Position
"O_SF_Rechtslauf"	M 439.1	BOOL	// M-AUSGANG: Rechtslauf Spaenefoerderer
"O_KM_Spruehpistole_ein"	M 439.2	BOOL	// M-AUSGANG: Pumpe Kühlmittel Spülpistole
"O_Spannhydraulik_Aus"	M 439.3	BOOL	// M-AUSGANG: Spannhydraulik entspannen
"O_AL_Blasluft_M25"	M 439.4	BOOL	// M-AUSGANG: Blasluft Kuehlung Werkzeug 'Ein'
"M_PW_Pumpe_Tischspuel"	M 439.5	BOOL	// PW: Palettenwechsler Pumpe Spülung
"M_SPI_LEITUNG_TEMP_RFG"	M 440.0	BOOL	// Spindel Leitungstemperatur: Reglerfreigabe
"M_VSP_Aktiv"	M 440.2	BOOL	// TEMPERATURKOMPENSATION: Vorsatzspindel aktiv
"O_Blasluft_Messtaster"	M 440.3	BOOL	// M-AUSGANG: Blasluft Messtaster
"M_M6_aktiv"	M 440.6	BOOL	// WZW: M6 aktiv
"M_M46_Gre_Hub_Grdst_Req"	M 440.7	BOOL	// WZW: Greifer / Hub Anforderung Grundstellung
"I_RPL_TASTE_DUSCHE_EIN"	M 441.0	BOOL	// ME G1-36.5 Bedienpult-RPL: Taste Spülung ein
"O_KM_RP_Dusche_Ventil"	M 441.1	BOOL	// MA G1-36.7 KM-Anlage Rüstplatz-Dusche Ventil Ein
"HM_PI_T_Spuelung_ein"	M 441.2	BOOL	// HM PI Rüstplatz Taste Spülung ein
"PI_RPT_T_Spuelung_ein"	M 441.3	BOOL	// PI Rüstplatz Taste Spülung ein
"O_RPL_KM_SPUELUNG_EIN"	M 441.4	BOOL	// MA xx-xx.x KM-Anlage Rüstplatz-Dusche Pumpe Ein
"M_KSA_Sammelfehler"	M 441.5	BOOL	// KSA3 Sammelfehler
"O_RPL_DUSCHE_EIN"	M 441.6	BOOL	// MA xx-xx.x KM-Anlage Rüstplatz-Dusche Meldelampe Ein
"O_Funktion_M180"	M 442.0	BOOL	// MZU: Ausgang M180
"O_Funktion_M181"	M 442.1	BOOL	// MZU: Ausgang M181
"O_Funktion_M182"	M 442.2	BOOL	// MZU: Ausgang M182
"O_Funktion_M183"	M 442.3	BOOL	// MZU: Ausgang M183
"O_Funktion_M184"	M 442.4	BOOL	// MZU: Ausgang M184
"O_Funktion_M185"	M 442.5	BOOL	// MZU: Ausgang M185
"O_Funktion_M186"	M 442.6	BOOL	// MZU: Ausgang M186
"O_Funktion_M187"	M 442.7	BOOL	// MZU: Ausgang M187
"O_Funktion_M188"	M 443.0	BOOL	// MZU: Ausgang M188
"O_Funktion_M189"	M 443.1	BOOL	// MZU: Ausgang M189
"O_KM_Pumpe_Dach"	M 443.2	BOOL	// M-AUSGANG: Spaenespuelung Dach
"O_KM_Spuelpumpe_ein"	M 443.3	BOOL	// M-AUSGANG: Spaenespuelung 'Ein'
"O_M7_Luftkuehlung"	M 443.4	BOOL	// M-AUSGANG: M7 Luftkuehlung
"O_KM_Pumpe_Dach2"	M 443.5	BOOL	// M-AUSGANG: Spaenespuelung 2 Dach
"O_WW_Rueck_MAG"	M 443.7	BOOL	// M-AUSGANG: Werkzeug-Rueckhalt ausfahren (verriegeln)
"O_WW_Hub_ZYL_in_Rein"	M 444.1	BOOL	// M-AUSGANG: Werkzeugreinigung zur Stellung Reinigen
"O_WW_Buersten_Reinigung"	M 444.3	BOOL	// M-AUSGANG: Antrieb Buerste Reinigung Werkzeugkegel
"I_ROBOT_LOCK"	M 444.4	BOOL	// ME F4-66.2 Schlüsselschalter Betriebsart Roboter gesperrt
"I_ROBOT_PROT_DOOR_CLSD"	M 444.5	BOOL	// ME F4-66.7 Werkstücklader Schutzzaun geschlossen
"O_Kab_Tuer_Entr"	M 444.7	BOOL	// M-AUSGANG: Lampe Taste Tuer Entriegeln
"O_LA_ausschwenken"	M 445.0	BOOL	// M-AUSGANG: Laser ausfahren
"O_LA_einschwenken"	M 445.1	BOOL	// M-AUSGANG: Laser einfahren
"O_LA_Sender_Ein"	M 445.2	BOOL	// M-AUSGANG: LaserFreigabe Sender
"O_LA_Empfaenger_Ein"	M 445.3	BOOL	// M-AUSGANG: Laser Freigabe Empänger
"O_LA_SCHMUTZB_AUF"	M 445.4	BOOL	// M-AUSGANG: Laser Ventil Schmutzblende
"O_LA_Sperrluft_Aus"	M 445.5	BOOL	// M-AUSGANG: Laser Ventil Sperrluft
"O_LA_ENABLE_EMPFAENGER2"	M 445.6	BOOL	// M-AUSGANG: Laser Freigabe Empänger 2
"O_WZK_Reinig_Blasluft"	M 446.0	BOOL	// M-AUSGANG: Werkzeugreinigung Blasluft
"I_GEN_OM_ID_SYNC"	M 446.1	BOOL	// M-EINGANG: Smartkey - Zeigt den START und RESTART der übertragung an (>50ms)
"I_GEN_OM_ID_CLOCK"	M 446.2	BOOL	// M-EINGANG: Smartkey - Protokoll-Taktrate. Daten können gelesen werden
"I_GEN_OM_ID_DATA_0"	M 446.3	BOOL	// M-EINGANG: Smartkey -  Daten-Spur 1
"I_GEN_OM_ID_DATA_1"	M 446.4	BOOL	// M-EINGANG: Smartkey -  Daten-Spur 2
"O_GEN_OM_ID_DATA_0"	M 446.5	BOOL	// M-AUSGANG: Smartkey -  Rückmeldung Daten-Spur 1
"O_GEN_OM_ID_DATA_1"	M 446.6	BOOL	// M-AUSGANG: Smartkey -  Rückmeldung Daten-Spur 2
"O_GEN_CNC_PGM_ACTIVE"	M 446.7	BOOL
"O_LA_WZ_ABBLASEN"	M 447.0	BOOL	// M-AUSGANG: Laser abblasen
"O_Y_Umschaltung_SPI"	M 447.1	BOOL	// M-AUSGANG: Stern Dreieck: Ausgang Stern
"O_D_Umschaltung_SPI"	M 447.2	BOOL	// M-AUSGANG: Stern Dreieck: Ausgang Dreieck
"O_PS_DREHST_BREMSE_AUF"	M 448.0	BOOL	// M-AUSGANG: Achse 9 (Palettenrundspeicher)  Bremse lüften
"O_PS_ABZIEHS_BREMSE_AUF"	M 448.1	BOOL	// M-AUSGANG: Bremse Kette 1 Palettenspeichersystem
"O_PS_RPL_BREMSE_AUF"	M 448.2	BOOL	// M-AUSGANG: Bremse Rüstplatz lüften
"O_PS_DREHST_HUB_AB"	M 448.3	BOOL	// M-AUSGANG: Ventil Dreheinheit nach unten
"O_PS_DREHST_HUB_AUF"	M 448.4	BOOL	// M-AUSGANG: Ventil Dreheinheit nach oben
"O_PS_RPL_TUER_VORN_ENTR"	M 448.5	BOOL	// M-AUSGANG: Ruestplatztuer vorn entriegeln
"O_PS_RPL_TUER_HINT_ENTR"	M 448.6	BOOL	// M-AUSGANG: Ruestplatztuer hinten entriegeln
"M_AchseNCT_loesen"	M 449.0	BOOL	// AX: NC-Teilapperat lösen
"M_AchseNCT_klemmen"	M 449.1	BOOL	// AX: NC-Teilapperat klemmen
"M_AchseNCT_Ready"	M 449.2	BOOL	// AX: NC-Teilapperat Ready mit klemmen / lösen
"M_AchseNCT_geloest"	M 449.3	BOOL	// AX: NC-Teilapperat gelöst
"M_A11_loes_aktiv"	M 449.4	BOOL	// AX: Achse 11 lösen aktiv
"I_D_PW_Tischspuelung"	M 450.0	BOOL	// M-EINGANG: Diagnose Spaenespülung Palettenwechsler
"I_D_KM_TPF_PAPIER_ENDE"	M 450.1	BOOL	// M-EINGANG: Diagnose Filterband Ende
"I_D_KM_TPF_PAPIER_WARN"	M 450.2	BOOL	// M-EINGANG: Diagnose Warnung Filterband Ende
"I_D_PW_HUB_IN_MITTE"	M 450.3	BOOL	// M-EINGANG: Palettenwechsler Diagnose Hub Pos. Mitte
"I_WW_POS_FRG_WZM"	M 450.4	BOOL	// M-EINGANG: Werkzeugwechsler Position Freigabe Werkzeugmagazin
"O_LED_Taste_Blau"	M 450.5	BOOL	// LED Taste Blau
"O_MessDose_Start"	M 450.6	BOOL	// M-AUSGANG: Laser Messdose ein
"O_WZ_MIN_SCH_MV1"	M 450.7	BOOL	// M-AUSGANG: Minimalmengen Schmierung Ventil 1 Ein
"O_AusBlasen_IKZ"	M 451.0	BOOL	// M-AUSGANG: Ausblasen IKZ Leitung
"O_AL_SCH_M26_Pumpe_ein"	M 451.1	BOOL	// M-AUSGANG: Dreh-Duchführung Ansteuerung Schmierpumpe 'Ein'
"M_SK_Sperre"	M 452.2	BOOL	// SCHWENKKOPF: Sperre
"Mx_FP_pos_Trigg_Blau"	M 453.0	BOOL	// LA:  FC_ZYLINDER Blaue Taste Flanke positiv
"Mx_FN_Blau"	M 453.1	BOOL	// LA:  FC_ZYLINDER Blaue Taste Flanke negativ
"Mx_Fp_GElb"	M 453.2	BOOL	// LA:  FC_ZYLINDER Gelbe Taste Flanke positiv
"Mx_Fn_Gelb"	M 453.3	BOOL	// LA:  FC_ZYLINDER Gelbe Taste Flanke negativ
"M_SSL_Aktiv"	M 453.7	BOOL	// WZV: NC Aktionssatz aktiv
"M_RPL_Bereich_1"	M 454.0	BOOL	// Rüstplatz Bereich 1
"M_RPL_Bereich_2"	M 454.1	BOOL	// Rüstplatz Bereich 2
"M_RPL_Bereich_3"	M 454.2	BOOL	// Rüstplatz Bereich 3
"M_RPL_Bereich_4"	M 454.3	BOOL	// Rüstplatz Bereich 4
"M_RPL_Pos_0"	M 454.4	BOOL	// Rüstplatz Position 0 Grad
"M_RPL_Pos_90"	M 454.5	BOOL	// Rüstplatz Position 90 Grad
"M_RPL_Pos_180"	M 454.6	BOOL	// Rüstplatz Position 180 Grad
"M_RPL_Pos_270"	M 454.7	BOOL	// Rüstplatz Position 270 Grad
"O_AL_ESR_AKTIV"	M 455.0	BOOL	// Rückmeldung Zyklus DM_ESR aktiv
"M_Wechsel_Prepare"	M 455.1	BOOL	// xxx
"M_T_WW_Gst_vorwaerts"	M 455.2	BOOL	// Taste Werkzeugwechsler vorwärts in Grundstellung fahren
"M_T_WW_Gst_rueckwaerts"	M 455.3	BOOL	// Taste Werkzeugwechsler rückwärts in Grundstellung fahren
"M_Tempkomp_eingefroren"	M 455.4	BOOL	// TEMPERATURKOMPENSATION: Eingefroren
"MX_IMP_W_Prep"	M 455.6	BOOL	// xxx
"MX_FP_W_Prep"	M 455.7	BOOL	// xxx
"M_out_mess_spindel"	M 456.0	BOOL	// xxx
"M_out_mess_spindel_2000"	M 456.1	BOOL	// xxx
"M_Not_aus"	M 456.3	BOOL	// MA: NOT-AUS  (*Maschine Ein)
"I_E_gerichtet"	M 456.4	BOOL	// M-EINGANG:
"I_WW_Y_inWWPos"	M 456.5	BOOL	// Y-Achse in Werkzeugwechselposition
"HM_PI_out_mess"	M 456.6	BOOL	// xxx
"PI_out_mess"	M 456.7	BOOL	// xxx
"O_AL_STILLSTAND"	M 457.0	BOOL	// M-AUSGANG: Stillstandueberwachung
"O_AL_NEG_NOTAUS"	M 457.1	BOOL	// M-AUSGANG: Not-Aus Drehzahl
"O_AL_TEST_BA"	M 457.2	BOOL	// Freigabe Drehzahl Betriebsarten
"I_WW_X_inWartePos"	M 457.4	BOOL	// X-Achse Werkzeugwechselwarteposition
"M_WW_Einzelfunktion"	M 457.5	BOOL	// xxx
"M_WW_Einzelschritt"	M 457.6	BOOL	// xxx
"I_WW_MagPlatz_frei"	M 457.7	BOOL	// M-EINGANG: Magazinplatz frei
"I_AL_5ACHS_KLE_GEKLEMMT"	M 458.0	BOOL	// M-EINGANG: Klemmung 5./11. Achse geklemmt
"O_KA2_STOERMELDUNG1"	M 458.1	BOOL	// M-AUSGANG: Kuehlaggregat 2 Störmeldung Prioritaet 1
"O_TA_KLEMMUNG_LOESEN"	M 458.2	BOOL	// M-AUSGANG: Klemmung loesen NC-Teilapparat
"O_SP_HYD_EIN"	M 458.3	BOOL	// M-AUSGANG: Spannhydraulik Pumpe ein
"O_WM_WZ_ZYL_CLAMP"	M 459.0	BOOL	// M-AUSGANG: Pneumatikzyl. Verriegelung WZ klemmen
"O_WM_WZ_ZYL_RELEASE"	M 459.1	BOOL	// M-AUSGANG: Pneumatikzylinder Verriegelung Werkzeug loesen
"I_WM_WZ_MAN_RELEASE"	M 459.2	BOOL	// M-EINGANG: Werkzeug manuell loesen
"O_WM_WZ_ZYL_RELEASE2"	M 459.3	BOOL	// M-AUSGANG: Pneumatikzylinder Verriegelung 2 Werkzeug loesen
"M_H5002_Wz_loesen"	M 459.4	BOOL	// WZW: H-Funktion 5002 Werkzeugspanner in Spindel lösen
"I_WK_SPINDEL_ABDECKUNG"	M 459.5	BOOL	// M-EINGANG: Spindel Abdeckung geschlossen
"MX_RefPkt_Achse"	M 460.0	BOOL	// AX6: (Spindel) Referenzpunkt Achse
"MX_Spdl_KorrWirksam"	M 460.1	BOOL	// AX6: (Spindel) Vorschubkorrektur wirksam setzen
"MX_Spdl_Spdl_Reset"	M 460.2	BOOL	// AX6: (Spindel) Spindel Reset
"MX_Spdl_Neu_Referenz"	M 460.3	BOOL	// AX6: (Spindel) neu Referieren
"MX_Spdl_Bei_Pos_NeuRef"	M 460.4	BOOL	// AX6: (Spindel) bei Positionieren neu Referieren
"MX_Spdl_RestwegLoeschen"	M 460.5	BOOL	// AX6: (Spindel) Restweg löschen
"I_SP_RPL_ALK_AUS"	M 460.6	BOOL	// ME H4-22.7 Schlüsselschalter Auflagekontrolle aus
"M_Req_GRF1_Mag"	M 460.7	BOOL	// WZW: Anforderung Greifer 1 zum Magazin
"MX_Spdl_PosBetr_84x5"	M 461.0	BOOL	// AX6: (Spindel) Positionierbetrieb
"MX_Spdl_DrehGrenz_83x0"	M 461.1	BOOL	// AX6: (Spindel) Drehzahlgrenze
"MX_Spdl_GewBohnre_84x3"	M 461.2	BOOL	// AX6: (Spindel) Gewindebohren aktiv
"MX_Spdl_SollBer_83x5"	M 461.3	BOOL	// AX6: (Spindel) Spindel im Sollbereich
"MX_Spdl_A_RefVerz_12x7"	M 461.4	BOOL	// AX6: (Spindel) Referenzverzögerung bei Motormessystem
"MX_Spdl_PendBetr_84x5"	M 461.5	BOOL	// AX6: (Spindel) Pendelbetrieb
"MX_Spdl_GetrUmsch_82x3"	M 461.6	BOOL	// AX6: (Spindel) Getriebeumschaltung 82x3
"MX_Spdl_E_RUCompl_94x2_"	M 461.7	BOOL	// AX6: (Spindel) Hochlauf beendet
"MX_Spdl_M3"	M 462.0	BOOL	// AX6: (Spindel) M3 (Rechtslauf) aktiv
"MX_Spdl_M4"	M 462.1	BOOL	// AX6: (Spindel) M4 (Linkslauf) aktiv
"MX_Spdl_M5"	M 462.2	BOOL	// AX6: (Spindel) M5 (Aus) aktiv
"MX_Spdl_M3_M4"	M 462.3	BOOL	// AX6: (Spindel) M3 oder M4 oder Fahrbefehl aktiv
"MX_Spdl_IMP_M3"	M 462.4	BOOL	// AX6: (Spindel) M3 (Rechtslauf) aktiv Impuls
"MX_Spdl_IMP_M4"	M 462.5	BOOL	// AX6: (Spindel) M4 (Linkslauf) aktiv Impuls
"MX_Spdl_IMP_M5"	M 462.6	BOOL	// AX6: (Spindel) M5 (Aus) aktiv Impuls
"MX_Spdl_IMP_M3_M4"	M 462.7	BOOL	// AX6: (Spindel) M3 oder M4 Impuls
"MX_Spdl_Reset_M3_4"	M 463.0	BOOL	// AX6: (Spindel) Reset M3 oder M4
"MX_Spdl_M3_Aktiv"	M 463.1	BOOL	// AX6: (Spindel) M3 (Rechtslauf) aktiv
"MX_Spdl_M4_Aktiv"	M 463.2	BOOL	// AX6: (Spindel) M3 (Linksslauf) aktiv
"MX_Spdl_FP_M4"	M 463.3	BOOL	// AX6: (Spindel) M4 (Linksslauf) aktiv Flanke positiv
"MX_Spdl_FP_M3"	M 463.4	BOOL	// AX6: (Spindel) M3 (Rechtslauf) aktiv Flanke positiv
"MX_Spdl_FP_M5"	M 463.5	BOOL	// AX6: (Spindel) M5 (Aus) aktiv Flanke positiv
"MX_Spdl_Hochlauf"	M 463.6	BOOL	// Spdl: Hochlauf nach Vorschub Halt
"MX_Spdl_Message_94x7"	M 463.7	BOOL	// AX6: (Spindel) Variable Meldefunktion
"MX_2GETR_VorFreig"	M 474.0	BOOL	// Getriebe: VorschubFreigabe
"MX_2Getr_AnfStufe"	M 474.1	BOOL	// Getriebe: Anforderung Stufe
"MX_2Getr_Aktiv"	M 474.2	BOOL	// Getriebe: Schalten Aktiv
"MX_2Getr_FP_Schalten"	M 474.3	BOOL	// Getriebe: Flanke Schalten
"MX_2Getr_FehlAus"	M 474.4	BOOL	// Getriebe: Fehler ausgegeben
"MX_Hawe_Ventil_0Sig"	M 474.5	BOOL	// Hawe Ventile Reitstock/Greifer 0Signal
"M_WZVS_M77_aktiviert"	M 474.6	BOOL	// WZVS mit M77 aktiviert
"Error_FC_SIEM_PLC_NCK"	M 474.7	BOOL	// Error-Meldung Baustein FC_SIEM_PLC_NCK
"I_MT_KAL_KLAPPE_ZU"	M 475.0	BOOL	// ME G5-14.3 Klappe Kalibriervorrichtung geschlossen
"I_MT_KALIBRIER_AUSG"	M 475.1	BOOL	// ME G5-14.5 Kalibrier Vorrichtung Messtaster ausgefahren
"I_MT_KALIBRIER_EING"	M 475.2	BOOL	// ME G5-14.6 Kalibrier Vorrichtung Messtaster eingefahren
"O_MT_KALIBRIER_AUSF"	M 475.3	BOOL	// MA G5-13.2 Kalibrier Vorrichtung Messtaster ausfahren
"O_MT_KALIBRIER_EINF"	M 475.4	BOOL	// MA G5-13.4 Kalibrier Vorrichtung Messtaster einfahren
"Mx_KSA_war_Aktiv"	M 475.5	BOOL	// Rückmeldung das ein M7,M8 angestanden hat
"Mx_Rauchnebel_fertig"	M 475.6	BOOL	// Rückmeldung Rauchnebelabscheider ist fertig
"mx_fn_rauchnebel"	M 475.7	BOOL	// Impuls für Rauchnebelabscheider
"M_SP_Vorschm_Req"	M 476.0	BOOL	// Spindelschmierung: Anforderung Vorschmierung
"M_WW_Bild_freifahren"	M 476.1	BOOL
"I_WW_MagTasche_auf"	M 476.2	BOOL	// M-EINGANG:
"I_WW_MagTasche_zu"	M 476.3	BOOL	// M-EINGANG:
"M_Vorschm_Imp_Ende"	M 476.4	BOOL
"M_Schmier_Imp_Ende"	M 476.5	BOOL
"M_SP_Nachschm_Req"	M 476.6	BOOL
"MX_IKZ_WZ_war_aktiv"	M 476.7	BOOL
"m_pw_schmier_stoe_dr_gsp"	M 477.0	BOOL	// Schmierung Palettenwechsler: Störung Druckaufbau gespeichert
"m_pw_start_aktiv_fp"	M 477.1	BOOL	// Palettenwechsler Start aktiv positive Flanke
"m_pw_Hub_Pos4_fn"	M 477.2	BOOL	// Position PW-Hub heben schnell
"m_pw_Hub_Pos4_fp"	M 477.3	BOOL	// Position PW-Hub senken schnell
"m_PWFG_unterdruecken"	M 477.4	BOOL	// Wegen "Schutzzaun-Funktionen" PW-Freigabe unterdruecken
"HM_PI_PWFG_unterdruecken"	M 477.5	BOOL	// HM PI Auslöser PW-Freigabe unterdrücken
"MX_FN_WZW_NC_Aktiv"	M 477.7	BOOL	// Flanke Negativ WZW NC aktiv
"IX_TLB_BIT_0"	M 500.0	BOOL	// M-EINGANG: WZB Binärcodiert
"IX_TLB_BIT_1"	M 500.1	BOOL	// M-EINGANG: WZB Binärcodiert
"IX_TLB_BIT_2"	M 500.2	BOOL	// M-EINGANG: WZB Binärcodiert
"IX_TLB_BIT_3"	M 500.3	BOOL	// M-EINGANG: WZB Binärcodiert
"IX_TLB_MEASURING_END"	M 500.4	BOOL	// M-EINGANG: WZB Messung Ende
"IX_TLB_HOME_POS"	M 500.5	BOOL	// M-EINGANG: WZB Parkstellung
"MX_Mag_Trigg4"	M 501.4	BOOL	// MAG: Trigger 4  (FC_MAG_HAUPT_ZH)
"MX_Mag_Trigg5"	M 501.5	BOOL	// MAG: Trigger 5  (FC_MAG_HAUPT_ZH)
"O_WM_Freigabe_re_li"	M 501.6	BOOL	// M-AUSGANG: Freigabe Werkzeugmagazin
"M_SK_Sicherpos"	M 503.0	BOOL
"M_AUTO_MAG_TOOL_RIEG_LOC"	M 504.0	BOOL
"M_AUTO_MAG_TOOL_RIEG_UNL"	M 504.1	BOOL
"M_K2_Programm_Aktiv"	M 504.2	BOOL
"M_K2_Vorschub_Halt"	M 504.3	BOOL
"I_TP_CALIBRATION_MOV_OU"	M 506.0	BOOL	// Messeinrichtung Messtaster ausgefahren
"I_TP_CALIBRATION_MOV_IN"	M 506.1	BOOL	// Messeinrichtung Messtaster eingefahren
"I_TP_CAL_FLAP_CLSD"	M 506.2	BOOL	// Klappe Messeinrichtung Geschlossen
"O_TP_CALIBRATION_EXTEND"	M 506.3	BOOL	// Messeinrichtung Messtaster ausfahren
"O_TP_CALIBRATION_RUN-IN"	M 506.4	BOOL	// Messeinrichtung Messtaster einfahren
"O_TP_CALIBRATION_CLEAN"	M 506.5	BOOL	// Messeinrichtung Messtaster abblasen
"MX_Ready_TM_TRANS"	M 507.0	BOOL
"M_H5000_H5004_WW_Start"	M 507.1	BOOL
"M_11Ax_plus"	M 510.0	BOOL
"M_11Ax_minus"	M 510.1	BOOL
"m_rqwwgf"	M 514.0	BOOL	// Autom.Grundstlg.fahren:Schritt Werkzeugwechsler Gf.
"m_rqpwgf"	M 514.1	BOOL	// Autom.Grundstlg.fahren:Schritt Palettenwechsler Gf.
"m_rqlagf"	M 514.2	BOOL	// Autom.Grundstlg.fahren: Schritt Laser Gf.
"M_LASER_IN_GRDST"	M 514.7	BOOL	// Laser Werkzeugvermessung in Grundstellung
"M_SO_DMS_PNEUMAK_EIN"	M 515.0	BOOL
"m_clrAl"	M 515.7	BOOL	// autom.Grundstlg.fahren:Reset Fehler/Meldungen
"M_FP_HubZyl_Start"	M 520.0	BOOL
"M_Fehl_WZB_Grdst"	M 520.1	BOOL
"M_Fehl_WZB_Grdst2"	M 520.2	BOOL
"M_FP_SPL_OK"	M 520.3	BOOL
"mx_fn_achs11"	M 520.7	BOOL
"I_KM_SF_KRATZ_NIV_MAX"	M 521.0	BOOL	// M-EINGANG: Max. Niveau-Überwachung  Kratzerförderer
"I_D_KM_SF_KRATZ_NIV_MAX"	M 521.1	BOOL	// M-EINGANG: Diagnose Max. Niveau-Überwachung  Kratzerförderer
"I_KM_SF_PUMPE_EIN"	M 521.2	BOOL	// M-EINGANG: Niveaukontrolle Schmutztank Hebepumpe „Ein“
"I_D_KM_SF_NEG_PUMPE_EIN"	M 521.3	BOOL	// M-EINGANG: Diagnose Niveau Schmutztank Hebepumpe „Ein“
"I_KM_SF_PUMPE_AUS"	M 521.4	BOOL	// M-EINGANG: Niveaukontrolle Schmutztank Hebepumpe „Aus“
"I_D_KM_SF_NEG_PUMPE_AUS"	M 521.5	BOOL	// M-EINGANG: Diagnose Niveau Schmutztank Hebepumpe „Aus“
"I_KM_SF_TANK_NIV_MAX"	M 521.6	BOOL	// M-EINGANG: Maximale Niveaukontrolle Schmutztank
"I_D_KM_SF_NEG_TANK_MAX"	M 521.7	BOOL	// M-EINGANG: Diagnose Maximale Niveaukontrolle Schmutztank
"I_TT_ausgeschwenkt"	M 522.0	BOOL	// M-EINGANG: Messtaster Tisch TS27R ausgeschwenkt
"I_TT_eingeschwenkt"	M 522.1	BOOL	// M-EINGANG: Messtaster Tisch TS27R eingeschwenkt
"O_KM_SF_KRATZER_EIN_V"	M 522.2	BOOL	// M-AUSGANG: Antrieb Kratzerförderer „Ein“
"O_KM_SF_HEBEPUMPE_EIN"	M 522.3	BOOL	// M-AUSGANG: Hebepumpe Schmutztank „Ein“
"O_AL_Messsignal_Umsch"	M 522.4	BOOL	// M-AUSGANG: Umschaltung Messsignale MesstasterTS27 / Laser
"O_TT_ausschwenken"	M 522.5	BOOL	// M-AUSGANG: Messtaster Tisch TS27R ausschwenken
"O_TT_einschwenken"	M 522.6	BOOL	// M-AUSGANG: Messtaster Tisch TS27R einschwenken
"O_TM_TPU_GET_TOOL"	M 523.0	BOOL	// M-AUSGANG: Transporteinheit auf Werkzeugkegel fahren
"I_TM_TPU_GET_TOOL"	M 523.1	BOOL	// M-EINGANG: Transporteinheit ist auf Werkzeugkegel gefahren
"O_TM_TPU_RELEASE_TOOL"	M 523.2	BOOL	// M-AUSGANG: Transporteinheit vom Werkzeugkegel wegfahren
"I_TM_TPU_RELEASE_TOOL"	M 523.3	BOOL	// M-EINGANG: Transporteinheit ist vom Werkzeugkegel weggefahren
"O_TM_TPU_TRANSFERPOS"	M 523.4	BOOL	// M-AUSGANG: Transporteinheit zu Übergabeposition fahren
"I_TM_TPU_TRANSFERPOS"	M 523.5	BOOL	// M-EINGANG: Transporteinheit ist zur Übergabeposition gefahren
"O_TM_TPU_MAGAZINPOS"	M 523.6	BOOL	// M-AUSGANG: Transporteinheit zur Magazinposition fahren
"I_TM_TPU_MAGAZINPOS"	M 523.7	BOOL	// M-EINGANG: Transporteinheit ist zur Magazinposition gefahren
"O_TM_MAG_TOOL_UNLOCK"	M 524.0	BOOL	// M-AUSGANG: Werkzeug an Magazinposition entriegeln
"I_TM_MAG_TOOL_UNLOCK"	M 524.1	BOOL	// M-EINGANG: Werkzeug an Magazinposition ist entriegelt (Zylinder)
"O_TM_MAG_TOOL_LOCK"	M 524.2	BOOL	// M-AUSGANG: Werkzeug an Magazinposition verriegeln
"I_TM_MAG_TOOL_LOCK"	M 524.3	BOOL	// M-EINGANG: Werkzeug an Magazinposition ist verriegelt (Zylinder)
"O_TM_TPU_AIR_CLEANING"	M 524.4	BOOL	// M-AUSGANG: Druckluftreinigung der Transporteinheit einschalten
"O_TM_TLOAD_TOOL_UNLOCK"	M 524.5	BOOL	// M-AUSGANG: Werkzeug am Rüstplatz entriegeln
"I_TM_TLOAD_TOOL_UNLOCK"	M 524.6	BOOL	// M-EINGANG: Werkzeug am Rüstplatz ist entriegelt (Zylinder)
"O_TM_TLOAD_TOOL_LOCK"	M 524.7	BOOL	// M-AUSGANG: Werkzeug am Rüstplatz verriegeln
"I_TM_TLOAD_TOOL_LOCK"	M 525.0	BOOL	// M-EINGANG: Werkzeug am Rüstplatz ist verriegelt (Zylinder)
"I_TM_TLOAD_PIN_LOCK"	M 525.1	BOOL	// M-EINGANG: Verriegelungspin Rüstplatz verriegelt (Kontrollschalter)
"I_TM_MAG_PIN_LOCK"	M 525.2	BOOL	// M-EINGANG: Verriegelungspin Magazinposition verriegelt (Kontrollschalter)
"M_SPI_belegt"	M 525.3	BOOL	// WZW: Werkzeug in der Spindel
"M_CU_Aktiv"	M 525.4	BOOL
"M_TPU_belegt"	M 525.5	BOOL
"M_Frg_WZ_vorbereiten"	M 525.6	BOOL
"M_Frg_WZ_ablegen"	M 525.7	BOOL
"M_WW_X_imArbeitsraum"	M 526.0	BOOL	// X-Achse im Arbeitsraum (bei Kettenmagazin)
"M_WZW_Transfer_Stellung"	M 526.1	BOOL
"NDR_WZDat_Lesen_2"	M 526.2	BOOL
"ERROR_WZDat_Lesen_2"	M 526.3	BOOL
"REQ_WZDat_Lesen_2"	M 526.4	BOOL
"I_TM_TLOAD_ACK_TOOL_IN"	M 526.5	BOOL
"I_TM_TLOAD_ACK_TOOL_OUT"	M 526.6	BOOL
"O_TM_TLOAD_TIN_H"	M 526.7	BOOL
"O_TM_TLOAD_TOUT_H"	M 527.0	BOOL
"M_Umsp_Wst_TPU"	M 527.1	BOOL
"M_Umsp_TPU_WST"	M 527.2	BOOL
"HM_PI_TM_VERW_1"	M 527.3	BOOL
"M_Umsp_Gr2_TPU"	M 527.4	BOOL
"HM_PI_TM_VERW_2"	M 527.5	BOOL
"M_Umsp_Gr1_TPU"	M 527.6	BOOL
"I_WW_X_inWWPos"	M 527.7	BOOL
"HM_PI_TM_VERW_3"	M 528.0	BOOL
"M_Umsp_TPU_Gr2"	M 528.1	BOOL
"HM_PI_TM_VERW_4"	M 528.2	BOOL
"M_AUTO_TPU_GET_TOOL"	M 528.3	BOOL
"M_AUTO_TPU_RELEASE_TOOL"	M 528.4	BOOL
"M_AUTO_TPU_MAGAZINPOS"	M 528.5	BOOL
"M_AUTO_TPU_TRANSFERPOS"	M 528.6	BOOL
"M_AUTO_MAG_TOOL_UNLOCK"	M 528.7	BOOL
"M_AUTO_MAG_TOOL_LOCK"	M 529.0	BOOL
"M_WZW_Fehler_Uebergabepl"	M 529.1	BOOL
"M_Schrittkette_Stop"	M 529.2	BOOL	// WZW: Schrittkette gestoppt durch Fehler
"M_WZW_SKZ_VOR"	M 529.3	BOOL
"M_WZW_FRG_SKZ_VOR"	M 529.4	BOOL
"M_WZW_SKZ_ZURUECK"	M 529.5	BOOL
"M_WZW_FRG_SKZ_ZURUECK"	M 529.6	BOOL
"M_WZW_GRDST_FAHRT_AKTIV"	M 529.7	BOOL
"M_FP_Greifer_drehen"	M 530.0	BOOL
"M_FN_Greifer_drehen"	M 530.1	BOOL
"M_PF_RF_X_Arbeitsraum"	M 530.2	BOOL
"M_PF_RF_X_WW_Pos"	M 530.3	BOOL
"M_PF_RF_Y_WW_Pos"	M 530.4	BOOL
"M_PF_RF_SPI_WW_Pos"	M 530.5	BOOL
"M_PF_RF_WW_180"	M 530.6	BOOL
"M_PF_RF_WW_360"	M 530.7	BOOL
"m_pWZWAsupAbbrechen"	M 531.0	BOOL	// WZW: Reset auslösen bei Abbruch Asup durch loslassen der Rettungs-Taste HM
"m_WZWAsupAbbrechen"	M 531.1	BOOL	// WZW: Reset auslösen bei Abbruch Asup durch loslassen der Rettungs-Taste
"M_FP_SKZ_VOR"	M 531.2	BOOL
"M_FP_SKZ_SAVE_RESET"	M 531.3	BOOL
"M_Frg_WW_Endstellung"	M 531.4	BOOL
"M_WW_Sperre_Wechsler"	M 531.5	BOOL
"Mx_Klappe_WZW_zu"	M 531.6	BOOL
"M_Greifer_rechts"	M 531.7	BOOL
"M_Greifer_links"	M 532.0	BOOL
"M_Grf1_0_Grad"	M 532.1	BOOL
"M_Grf1_180_Grad"	M 532.2	BOOL
"M_FN_Greifer drehen"	M 532.3	BOOL
"M_FP_SKZ_ZURUECK"	M 532.4	BOOL
"M_FP_Grf1_0_Grad"	M 532.5	BOOL
"M_FP_Grf1_180_Grad"	M 532.6	BOOL
"M_AUTO_TLOAD_TOOL_LOCK"	M 532.7	BOOL
"M_AUTO_TLOAD_TOOL_UNLOCK"	M 533.0	BOOL
"M_SperreMag_Wz_einlegen"	M 533.1	BOOL
"M_VSP_Mag_Vertikalkette"	M 533.2	BOOL
"I_DM_Ta_NC-Start"	M 533.3	BOOL
"I_WWT_offen"	M 533.4	BOOL
"I_WMT_verriegelt"	M 533.5	BOOL
"I_TM_TLOAD_TOOL_INSERT"	M 533.6	BOOL	// M-EINGANG: Positionsüberwachung Werkzeug Rüstplatz
"M_MTH_READY_SOKO"	M 534.0	BOOL
"I_PS_RPL_DREHZAHL_BIT_1"	M 534.4	BOOL	// Drehzahl Ruestplatz binaer codiert 2\20
"I_PS_RPL_DREHZAHL_BIT_2"	M 534.5	BOOL	// Drehzahl Ruestplatz binaer codiert 2\21
"I_PS_RPL_DREHZAHL_BIT_3"	M 534.6	BOOL	// Drehzahl Ruestplatz binaer codiert 2\22
"I_PS_RPL_DREHZAHL_BIT_4"	M 534.7	BOOL	// Drehzahl Ruestplatz binaer codiert 2\23
"m_request_qeifer_WZ_Gr"	M 535.0	BOOL	// Request lesen Greifer OEM Daten
"M_WZ_Wasch_schnell"	M 535.1	BOOL	// Wz Waschen 1 Sekunde aus Wz Verwaltung
"M_WZ_Wasch_abgewaehlt"	M 535.2	BOOL	// Waschen von WZ verwaltung abgewählt
"m_FLM_request_read"	M 535.3	BOOL	// FLM fuer Lesen Greifer OEM Daten
"m_VSH_SP_GETRIEBE"	M 535.4	BOOL	// Vorschubhalt von Ueberwachung Getriebeumschaltung Spindel
"O_WK_MAG_AUSFAHREN"	M 535.5	BOOL	// Werkzeugtraeger ausfahren
"O_WK_MAG_EINFAHREN"	M 535.6	BOOL	// Werkzeugtraeger einfahren
"I_WK_GRUNDSTELL"	M 535.7	BOOL	// Werkzeugtraeger Grundstellung
"I_WK_WECH_POS"	M 536.0	BOOL	// Werkzeugtraeger Wechselposition
"O_WK_ZYL_2_AUSF"	M 536.1	BOOL	// Werkzeugtraeger Zylinder 2 ausfahren
"O_WK_ZYL_2_EINFAHREN"	M 536.2	BOOL	// Werkzeugtraeger Zylinder 2 einfahren
"I_WK_ZYL_2_GST"	M 536.3	BOOL	// Werkzeugtraeger Zylinder 2 Grundstellung
"I_WK_ZYL_2_WE_POS"	M 536.4	BOOL	// Werkzeugtraeger Zylinder 2 Wechselposition
"O_WK_KLAPPE_AUF"	M 536.5	BOOL	// Werkzeugklappe oeffnen
"O_WK_KLAPPE_ZU"	M 536.6	BOOL	// Werkzeugklappe schliessen
"I_WK_KLAPPE_AUF"	M 536.7	BOOL	// Werkzeugklappe geoeffnet
"I_WK_KLAPPE_ZU"	M 537.0	BOOL	// Werkzeugklappe geschlossen
"I_WK_WZ_1_VORHANDEN"	M 537.1	BOOL	// Winkelfraeskopf 1 vorhanden
"I_WK_WZ_2_VORHANDEN"	M 537.2	BOOL	// Winkelfraeskopf 2 vorhanden
"M_VSH_GetrUeberw_aktiv"	M 537.7	BOOL	// Vorschub-Halt Überwachung Getriebeumschaltung aktiv (gespeichert)
"M_WK_Auto_Klappe_oeffnen"	M 538.0	BOOL
"M_WK_Auto_Pos1_AST"	M 538.1	BOOL
"M_WK_Auto_Pos2_AST"	M 538.2	BOOL
"M_WK_Auto_Grdst"	M 538.3	BOOL
"M_WK_Auto_Zyl2_Grdst"	M 538.4	BOOL
"M_WK_Auto_Klappe_schlies"	M 538.5	BOOL
"M_WIKO_Asup_abbrechen"	M 538.6	BOOL	// WIKO: Reset auslösen bei Abbruch Asup durch loslassen der Rettungs-Taste
"M_PW_Asup_abbrechen"	M 538.7	BOOL	// PW: Reset auslösen bei Abbruch Asup durch loslassen der Rettungs-Taste
"M_SBH_AKTIV_ARBEITSRAUM"	M 539.0	BOOL	// SAFETY: SBH aktiv -> Freigabe Arbeitsraumtüre entriegeln
"M_SBH_AKTIV_RÜSTPLATZ"	M 539.1	BOOL	// SAFETY: SBH aktiv -> Freigabe Rüstplatztüre Palettenwechsler entriegeln
"M_SBH_AKTIV_MAGAZIN"	M 539.2	BOOL	// SAFETY: SBH aktiv -> Freigabe Magazintüre entriegeln
"M_SBH_AKTIV_RPL_PS"	M 539.3	BOOL	// SAFETY: SBH aktiv -> Freigabe Rüstplatztüre Palettenspeicher entriegeln
"M_SBH_ANF_ARBEITSRAUM"	M 539.4	BOOL	// SAFETY: SBH Anforderung Arbeitsraum
"M_SBH_ANF_RÜSTPLATZ"	M 539.5	BOOL	// SAFETY: SBH Anforderung Palettenwechsler
"M_SBH_ANF_MAGAZIN"	M 539.6	BOOL	// SAFETY: SBH Anforderung Magazin
"M_SBH_ANF_RPL_PS"	M 539.7	BOOL	// SAFETY: SBH Anforderung  Palettenspeicher
"M_Umsp_TPU_Gr1"	M 540.0	BOOL
"M_FN_RP_Palette_weg"	M 540.1	BOOL
"M_FN_RP_Pal_auf_0"	M 540.2	BOOL
"M_Kegelrein_VM_aktiv"	M 540.3	BOOL
"M_Anwahl_WZW_Maske"	M 540.7	BOOL	// Anwahl für Maske Schneller Werkzeugwechsel
"I_TM_TOOL_CYL_LOCKED"	M 541.0	BOOL
"I_TM_TOOL_CYL_UNLOCKED"	M 541.1	BOOL
"M_AUTO_TLOAD_CYL_LOCK"	M 541.2	BOOL
"M_AUTO_TLOAD_CYL_UNLOCK"	M 541.3	BOOL
"O_TM_TOOL_CYL_LOCK"	M 541.4	BOOL
"M_FP_Auto_TLoad_Tool_Loc"	M 541.5	BOOL
"M_FN_Te_Pin_Ruest_Lock"	M 541.6	BOOL
"M_FP_TLOAD_TOOL_LOCK"	M 541.7	BOOL
"m_oem_freigabe_bew_nr"	M 549.0	BOOL	// OEM: Freigabe OEM Bewegungsnummer (Taste Blau/Gelb aktiv)
"m_oem_reset_frg_bew_nr"	M 549.1	BOOL	// OEM: Reset Freigabe OEM Bewegungsnummer Flanke Positiv
"M_FP_Achse14_steht"	M 549.2	BOOL
"M_FP_Achse_WZGR_Pos_lese"	M 549.3	BOOL
"M_FP_Einlesesperre"	M 549.7	BOOL
"m_hmi_pro_taste_plus"	M 550.0	BOOL	// HMI-PRO: Taste plus
"m_hmi_pro_taste_minus"	M 550.1	BOOL	// HMI-PRO: Taste minus
"m_550.2"	M 550.2	BOOL	// HMI-PRO:
"m_550.3"	M 550.3	BOOL	// HMI-PRO:
"m_550.4"	M 550.4	BOOL	// HMI-PRO:
"m_550.5"	M 550.5	BOOL	// HMI-PRO:
"m_550.6"	M 550.6	BOOL	// HMI-PRO:
"m_550.7"	M 550.7	BOOL	// HMI-PRO:
"m_hmi_pro_m551.0"	M 551.0	BOOL	// HMI-PRO: Bild Einschaltbedingungen -
"m_hmi_pro_m551.1"	M 551.1	BOOL	// HMI-PRO: Bild Einschaltbedingungen -
"m_hmi_pro_HYD_einschalt"	M 551.2	BOOL	// HMI-PRO: Bild Einschaltbedingungen -  Hydraulik EIN
"m_hmi_pro_HYD_ausschalt"	M 551.3	BOOL	// HMI-PRO: Bild Einschaltbedingungen -  Hydraulik AUS
"m_hmi_pro_PNEU_einschalt"	M 551.4	BOOL	// HMI-PRO: Bild Einschaltbedingungen -  Pneumatik EIN
"m_hmi_pro_PNEU_ausschalt"	M 551.5	BOOL	// HMI-PRO: Bild Einschaltbedingungen -  Pneumatik AUS
"m_hmi_pro_KMTL_einschalt"	M 551.6	BOOL	// HMI-PRO: Bild Einschaltbedingungen -  Kühlmitelanlage EIN
"m_hmi_pro_KMTL_ausschalt"	M 551.7	BOOL	// HMI-PRO: Bild Einschaltbedingungen -  Kühlmitelanlage AUS
"m_552.0"	M 552.0	BOOL	// HMI-PRO:
"m_552.1"	M 552.1	BOOL	// HMI-PRO:
"m_552.2"	M 552.2	BOOL	// HMI-PRO:
"m_552.3"	M 552.3	BOOL	// HMI-PRO:
"m_552.4"	M 552.4	BOOL	// HMI-PRO:
"m_552.5"	M 552.5	BOOL	// HMI-PRO:
"m_552.6"	M 552.6	BOOL	// HMI-PRO:
"m_552.7"	M 552.7	BOOL	// HMI-PRO:
"m_hmi_pro_HYD_ein_gesp"	M 553.0	BOOL	// HMI-PRO: Bild Einschaltbedingungen - Hydraulik EIN gespeichert
"m_hmi_pro_PNEU_ein_gesp"	M 553.1	BOOL	// HMI-PRO: Bild Einschaltbedingungen - Pneumatik EIN gespeichert
"m_553.2"	M 553.2	BOOL	// HMI-PRO:
"m_553.3"	M 553.3	BOOL	// HMI-PRO:
"m_553.4"	M 553.4	BOOL	// HMI-PRO:
"m_553.5"	M 553.5	BOOL	// HMI-PRO:
"m_553.6"	M 553.6	BOOL	// HMI-PRO:
"m_553.7"	M 553.7	BOOL	// HMI-PRO:
"m_hmi_pro_zeile_mb554.0"	M 554.0	BOOL	// HMI-PRO: Byte Einrichtzeilennummer
"m_hmi_pro_zeile_mb554.1"	M 554.1	BOOL	// HMI-PRO: Byte Einrichtzeilennummer
"m_hmi_pro_zeile_mb554.2"	M 554.2	BOOL	// HMI-PRO: Byte Einrichtzeilennummer
"m_hmi_pro_zeile_mb554.3"	M 554.3	BOOL	// HMI-PRO: Byte Einrichtzeilennummer
"m_hmi_pro_zeile_mb554.4"	M 554.4	BOOL	// HMI-PRO: Byte Einrichtzeilennummer
"m_hmi_pro_zeile_mb554.5"	M 554.5	BOOL	// HMI-PRO: Byte Einrichtzeilennummer
"m_hmi_pro_zeile_mb554.6"	M 554.6	BOOL	// HMI-PRO: Byte Einrichtzeilennummer
"m_hmi_pro_zeile_mb554.7"	M 554.7	BOOL	// HMI-PRO: Byte Einrichtzeilennummer
"m_hmi_pro_m555.0"	M 555.0	BOOL	// HMI-PRO: Taktart -
"m_hmi_pro_leerfahren_akt"	M 555.1	BOOL	// HMI-PRO: Taktart - Leerfahren aktiv
"m_hmi_pro_warmfahren_akt"	M 555.2	BOOL	// HMI-PRO: Taktart - Warmfahren aktiv
"m_hmi_pro_fahren_oW_akt"	M 555.3	BOOL	// HMI-PRO: Taktart - Fahren ohne Werkstück aktiv
"m_555.4"	M 555.4	BOOL	// HMI-PRO: Taktart -
"m_555.5"	M 555.5	BOOL	// HMI-PRO: Taktart -
"m_555.6"	M 555.6	BOOL	// HMI-PRO: Taktart -
"m_555.7"	M 555.7	BOOL	// HMI-PRO: Taktart -
"m_556.0"	M 556.0	BOOL	// HMI-PRO:
"m_556.1"	M 556.1	BOOL	// HMI-PRO:
"m_556.2"	M 556.2	BOOL	// HMI-PRO:
"m_556.3"	M 556.3	BOOL	// HMI-PRO:
"m_556.4"	M 556.4	BOOL	// HMI-PRO:
"m_556.5"	M 556.5	BOOL	// HMI-PRO:
"m_556.6"	M 556.6	BOOL	// HMI-PRO:
"m_556.7"	M 556.7	BOOL	// HMI-PRO:
"m_557.0"	M 557.0	BOOL	// HMI-PRO:
"m_557.1"	M 557.1	BOOL	// HMI-PRO:
"m_557.2"	M 557.2	BOOL	// HMI-PRO:
"m_557.3"	M 557.3	BOOL	// HMI-PRO:
"m_557.4"	M 557.4	BOOL	// HMI-PRO:
"m_557.5"	M 557.5	BOOL	// HMI-PRO:
"m_557.6"	M 557.6	BOOL	// HMI-PRO:
"m_557.7"	M 557.7	BOOL	// HMI-PRO:
"m_558.0"	M 558.0	BOOL	// HMI-PRO:
"m_558.1"	M 558.1	BOOL	// HMI-PRO:
"m_558.2"	M 558.2	BOOL	// HMI-PRO:
"m_558.3"	M 558.3	BOOL	// HMI-PRO:
"m_558.4"	M 558.4	BOOL	// HMI-PRO:
"m_558.5"	M 558.5	BOOL	// HMI-PRO:
"m_558.6"	M 558.6	BOOL	// HMI-PRO:
"m_558.7"	M 558.7	BOOL	// HMI-PRO:
"m_559.0"	M 559.0	BOOL	// HMI-PRO:
"m_559.1"	M 559.1	BOOL	// HMI-PRO:
"m_559.2"	M 559.2	BOOL	// HMI-PRO:
"m_559.3"	M 559.3	BOOL	// HMI-PRO:
"m_559.4"	M 559.4	BOOL	// HMI-PRO:
"m_559.5"	M 559.5	BOOL	// HMI-PRO:
"m_559.6"	M 559.6	BOOL	// HMI-PRO:
"m_559.7"	M 559.7	BOOL	// HMI-PRO:
"MX_Error_RD_IstPos14"	M 560.0	BOOL	// HMI-PRO:
"MX_NDR_RD_IstPos14"	M 560.1	BOOL	// HMI-PRO:
"m_560.2"	M 560.2	BOOL	// HMI-PRO:
"m_560.3"	M 560.3	BOOL	// HMI-PRO:
"m_560.4"	M 560.4	BOOL	// HMI-PRO:
"m_560.5"	M 560.5	BOOL	// HMI-PRO:
"m_560.6"	M 560.6	BOOL	// HMI-PRO:
"m_560.7"	M 560.7	BOOL	// HMI-PRO:
"m_561.0"	M 561.0	BOOL	// HMI-PRO:
"m_561.1"	M 561.1	BOOL	// HMI-PRO:
"m_561.2"	M 561.2	BOOL	// HMI-PRO:
"m_561.3"	M 561.3	BOOL	// HMI-PRO:
"m_561.4"	M 561.4	BOOL	// HMI-PRO:
"m_561.5"	M 561.5	BOOL	// HMI-PRO:
"m_561.6"	M 561.6	BOOL	// HMI-PRO:
"m_561.7"	M 561.7	BOOL	// HMI-PRO:
"m_562.0"	M 562.0	BOOL	// HMI-PRO:
"m_562.1"	M 562.1	BOOL	// HMI-PRO:
"m_562.2"	M 562.2	BOOL	// HMI-PRO:
"m_562.3"	M 562.3	BOOL	// HMI-PRO:
"m_562.4"	M 562.4	BOOL	// HMI-PRO:
"m_562.5"	M 562.5	BOOL	// HMI-PRO:
"m_562.6"	M 562.6	BOOL	// HMI-PRO:
"m_562.7"	M 562.7	BOOL	// HMI-PRO:
"m_563.0"	M 563.0	BOOL	// HMI-PRO:
"m_563.1"	M 563.1	BOOL	// HMI-PRO:
"m_563.2"	M 563.2	BOOL	// HMI-PRO:
"m_563.3"	M 563.3	BOOL	// HMI-PRO:
"m_563.4"	M 563.4	BOOL	// HMI-PRO:
"m_563.5"	M 563.5	BOOL	// HMI-PRO:
"m_563.6"	M 563.6	BOOL	// HMI-PRO:
"m_563.7"	M 563.7	BOOL	// HMI-PRO:
"m_564.0"	M 564.0	BOOL	// HMI-PRO:
"m_564.1"	M 564.1	BOOL	// HMI-PRO:
"m_564.2"	M 564.2	BOOL	// HMI-PRO:
"m_564.3"	M 564.3	BOOL	// HMI-PRO:
"m_564.4"	M 564.4	BOOL	// HMI-PRO:
"m_564.5"	M 564.5	BOOL	// HMI-PRO:
"m_564.6"	M 564.6	BOOL	// HMI-PRO:
"m_564.7"	M 564.7	BOOL	// HMI-PRO:
"m_565.0"	M 565.0	BOOL	// HMI-PRO:
"m_565.1"	M 565.1	BOOL	// HMI-PRO:
"m_565.2"	M 565.2	BOOL	// HMI-PRO:
"m_565.3"	M 565.3	BOOL	// HMI-PRO:
"m_565.4"	M 565.4	BOOL	// HMI-PRO:
"m_565.5"	M 565.5	BOOL	// HMI-PRO:
"m_565.6"	M 565.6	BOOL	// HMI-PRO:
"m_565.7"	M 565.7	BOOL	// HMI-PRO:
"m_566.0"	M 566.0	BOOL	// HMI-PRO:
"m_566.1"	M 566.1	BOOL	// HMI-PRO:
"m_566.2"	M 566.2	BOOL	// HMI-PRO:
"m_566.3"	M 566.3	BOOL	// HMI-PRO:
"m_566.4"	M 566.4	BOOL	// HMI-PRO:
"m_566.5"	M 566.5	BOOL	// HMI-PRO:
"m_566.6"	M 566.6	BOOL	// HMI-PRO:
"m_566.7"	M 566.7	BOOL	// HMI-PRO:
"m_567.0"	M 567.0	BOOL	// HMI-PRO:
"m_567.1"	M 567.1	BOOL	// HMI-PRO:
"m_567.2"	M 567.2	BOOL	// HMI-PRO:
"m_567.3"	M 567.3	BOOL	// HMI-PRO:
"m_567.4"	M 567.4	BOOL	// HMI-PRO:
"m_567.5"	M 567.5	BOOL	// HMI-PRO:
"m_567.6"	M 567.6	BOOL	// HMI-PRO:
"m_567.7"	M 567.7	BOOL	// HMI-PRO:
"m_568.0"	M 568.0	BOOL	// HMI-PRO:
"m_568.1"	M 568.1	BOOL	// HMI-PRO:
"m_568.2"	M 568.2	BOOL	// HMI-PRO:
"m_568.3"	M 568.3	BOOL	// HMI-PRO:
"m_568.4"	M 568.4	BOOL	// HMI-PRO:
"m_568.5"	M 568.5	BOOL	// HMI-PRO:
"m_568.6"	M 568.6	BOOL	// HMI-PRO:
"m_568.7"	M 568.7	BOOL	// HMI-PRO:
"m_569.0"	M 569.0	BOOL	// HMI-PRO:
"m_569.1"	M 569.1	BOOL	// HMI-PRO:
"m_569.2"	M 569.2	BOOL	// HMI-PRO:
"m_569.3"	M 569.3	BOOL	// HMI-PRO:
"m_569.4"	M 569.4	BOOL	// HMI-PRO:
"m_569.5"	M 569.5	BOOL	// HMI-PRO:
"m_569.6"	M 569.6	BOOL	// HMI-PRO:
"m_569.7"	M 569.7	BOOL	// HMI-PRO:
"m_572.0"	M 572.0	BOOL	// HMI-PRO:
"m_572.1"	M 572.1	BOOL	// HMI-PRO:
"m_572.2"	M 572.2	BOOL	// HMI-PRO:
"m_572.3"	M 572.3	BOOL	// HMI-PRO:
"m_572.4"	M 572.4	BOOL	// HMI-PRO:
"m_572.5"	M 572.5	BOOL	// HMI-PRO:
"m_572.6"	M 572.6	BOOL	// HMI-PRO:
"m_572.7"	M 572.7	BOOL	// HMI-PRO:
"m_573.0"	M 573.0	BOOL	// HMI-PRO:
"m_573.1"	M 573.1	BOOL	// HMI-PRO:
"m_573.2"	M 573.2	BOOL	// HMI-PRO:
"m_573.3"	M 573.3	BOOL	// HMI-PRO:
"m_573.4"	M 573.4	BOOL	// HMI-PRO:
"m_573.5"	M 573.5	BOOL	// HMI-PRO:
"m_573.6"	M 573.6	BOOL	// HMI-PRO:
"m_573.7"	M 573.7	BOOL	// HMI-PRO:
"m_574.0"	M 574.0	BOOL	// HMI-PRO:
"m_574.1"	M 574.1	BOOL	// HMI-PRO:
"m_574.2"	M 574.2	BOOL	// HMI-PRO:
"m_574.3"	M 574.3	BOOL	// HMI-PRO:
"m_574.4"	M 574.4	BOOL	// HMI-PRO:
"m_574.5"	M 574.5	BOOL	// HMI-PRO:
"m_574.6"	M 574.6	BOOL	// HMI-PRO:
"m_574.7"	M 574.7	BOOL	// HMI-PRO:
"m_575.0"	M 575.0	BOOL	// HMI-PRO:
"m_575.1"	M 575.1	BOOL	// HMI-PRO:
"m_575.2"	M 575.2	BOOL	// HMI-PRO:
"m_575.3"	M 575.3	BOOL	// HMI-PRO:
"m_575.4"	M 575.4	BOOL	// HMI-PRO:
"m_575.5"	M 575.5	BOOL	// HMI-PRO:
"m_575.6"	M 575.6	BOOL	// HMI-PRO:
"m_575.7"	M 575.7	BOOL	// HMI-PRO:
"m_576.0"	M 576.0	BOOL	// HMI-PRO:
"m_576.1"	M 576.1	BOOL	// HMI-PRO:
"m_576.2"	M 576.2	BOOL	// HMI-PRO:
"m_576.3"	M 576.3	BOOL	// HMI-PRO:
"m_576.4"	M 576.4	BOOL	// HMI-PRO:
"m_576.5"	M 576.5	BOOL	// HMI-PRO:
"m_576.6"	M 576.6	BOOL	// HMI-PRO:
"m_576.7"	M 576.7	BOOL	// HMI-PRO:
"m_577.0"	M 577.0	BOOL	// HMI-PRO:
"m_577.1"	M 577.1	BOOL	// HMI-PRO:
"m_577.2"	M 577.2	BOOL	// HMI-PRO:
"m_577.3"	M 577.3	BOOL	// HMI-PRO:
"m_577.4"	M 577.4	BOOL	// HMI-PRO:
"m_577.5"	M 577.5	BOOL	// HMI-PRO:
"m_577.6"	M 577.6	BOOL	// HMI-PRO:
"m_577.7"	M 577.7	BOOL	// HMI-PRO:
"m_578.0"	M 578.0	BOOL	// HMI-PRO:
"m_578.1"	M 578.1	BOOL	// HMI-PRO:
"m_578.2"	M 578.2	BOOL	// HMI-PRO:
"m_578.3"	M 578.3	BOOL	// HMI-PRO:
"m_578.4"	M 578.4	BOOL	// HMI-PRO:
"m_578.5"	M 578.5	BOOL	// HMI-PRO:
"m_578.6"	M 578.6	BOOL	// HMI-PRO:
"m_578.7"	M 578.7	BOOL	// HMI-PRO:
"m_579.0"	M 579.0	BOOL	// HMI-PRO:
"m_579.1"	M 579.1	BOOL	// HMI-PRO:
"m_579.2"	M 579.2	BOOL	// HMI-PRO:
"m_579.3"	M 579.3	BOOL	// HMI-PRO:
"m_579.4"	M 579.4	BOOL	// HMI-PRO:
"m_579.5"	M 579.5	BOOL	// HMI-PRO:
"m_579.6"	M 579.6	BOOL	// HMI-PRO:
"m_579.7"	M 579.7	BOOL	// HMI-PRO:
"m_hmi_mdebde_start_gesp"	M 580.0	BOOL	// HMI-PRO: MDEBDE Start eingeleitet gespeichert
"m_hmi_sofort_halt_gesp"	M 580.1	BOOL	// HMI-PRO: <Sofort Halt> gespeichert
"m_hmi_prisma_wkst_zaehl"	M 580.2	BOOL	// HMI-PRO: Prisma: Werkstückzähltakt
"m_hmi_prisma_zaehl_fp"	M 580.3	BOOL	// HMI-PRO: Werkstückzählung Zähltakt Flanke positiv
"m_hmi_taktzeit_ges"	M 581.0	BOOL	// HMI-PRO: Taktzeitmessung Gesamt
"m_hmi_taktzeit_ges_fp1"	M 581.1	BOOL	// HMI-PRO: Taktzeitmessung Gesamt Flanke positiv 1
"m_hmi_taktzeit_ges_fp2"	M 581.2	BOOL	// HMI-PRO: Taktzeitmessung Gesamt Flanke positiv 2
"m_hmi_taktzeit_ges_hm"	M 581.3	BOOL	// HMI-PRO: Taktzeitmessung Gesamt Hilfsmerker
"m_hmi_taktzeit_pw"	M 581.4	BOOL	// HMI-PRO: Taktzeitmessung Palettenwechsler
"m_hmi_taktzeit_pw_fp1"	M 581.5	BOOL	// HMI-PRO: Taktzeitmessung PalettenwechslerFlanke positiv 1
"m_hmi_taktzeit_pw_fp2"	M 581.6	BOOL	// HMI-PRO: Taktzeitmessung PalettenwechslerFlanke positiv 2
"m_hmi_taktzeit_pw_hm"	M 581.7	BOOL	// HMI-PRO: Taktzeitmessung PalettenwechslerHilfsmerker
"m_hmi_taktzeit_masch"	M 582.0	BOOL	// HMI-PRO: Taktzeitmessung Maschine
"m_hmi_taktzeit_masch_fp1"	M 582.1	BOOL	// HMI-PRO: Taktzeitmessung MaschineFlanke positiv 1
"m_hmi_taktzeit_masch_fp2"	M 582.2	BOOL	// HMI-PRO: Taktzeitmessung MaschineFlanke positiv 2
"m_hmi_taktzeit_masch_hm"	M 582.3	BOOL	// HMI-PRO: Taktzeitmessung MaschineHilfsmerker
"m_hmi_lampentest_fn"	M 582.4	BOOL	// HMI-PRO: Lampentest negative Flanke
"m_hmi_nc_start_led_hm"	M 582.5	BOOL	// HMI-PRO: LED NC Start Hilfsmerker
"I_DirektTaste_1_links"	M 588.0	BOOL	// HMI-PRO: OP12/OP15A Direkttaste 1 links
"I_DirektTaste_2_links"	M 588.1	BOOL	// HMI-PRO: OP12/OP15A Direkttaste 2 links
"I_DirektTaste_3_links"	M 588.2	BOOL	// HMI-PRO: OP12/OP15A Direkttaste 3 links
"I_DirektTaste_4_links"	M 588.3	BOOL	// HMI-PRO: OP12/OP15A Direkttaste 4 links
"I_DirektTaste_5_links"	M 588.4	BOOL	// HMI-PRO: OP12/OP15A Direkttaste 5 links
"I_DirektTaste_6_links"	M 588.5	BOOL	// HMI-PRO: OP12/OP15A Direkttaste 6 links
"I_DirektTaste_7_links"	M 588.6	BOOL	// HMI-PRO: OP12/OP15A Direkttaste 7 links
"I_DirektTaste_8_links"	M 588.7	BOOL	// HMI-PRO: OP12/OP15A Direkttaste 8 links
"I_DirektTaste_1_rechts"	M 589.0	BOOL	// HMI-PRO: OP12/OP15A Direkttaste 1 rechts
"I_DirektTaste_2_rechts"	M 589.1	BOOL	// HMI-PRO: OP12/OP15A Direkttaste 2 rechts
"I_DirektTaste_3_rechts"	M 589.2	BOOL	// HMI-PRO: OP12/OP15A Direkttaste 3 rechts
"I_DirektTaste_4_rechts"	M 589.3	BOOL	// HMI-PRO: OP12/OP15A Direkttaste 4 rechts
"I_DirektTaste_5_rechts"	M 589.4	BOOL	// HMI-PRO: OP12/OP15A Direkttaste 5 rechts
"I_DirektTaste_6_rechts"	M 589.5	BOOL	// HMI-PRO: OP12/OP15A Direkttaste 6 rechts
"I_DirektTaste_7_rechts"	M 589.6	BOOL	// HMI-PRO: OP12/OP15A Direkttaste 7 rechts
"I_DirektTaste_8_rechts"	M 589.7	BOOL	// HMI-PRO: OP12/OP15A Direkttaste 8 rechts
"m_tueren_ges_geschl+verr"	M 590.0	BOOL	// TL2000: Schutztüren gesamt geschlossen und verriegelt
"Mx_ReqKlemm_Grundzustand"	M 590.1	BOOL	// Klemmungsgrundzustand bei erstem Verfahrbefehl(früher bei RESET)
"m_590.2"	M 590.2	BOOL	// TL2000:
"m_590.3"	M 590.3	BOOL	// TL2000:
"m_590.4"	M 590.4	BOOL	// TL2000:
"m_590.5"	M 590.5	BOOL	// TL2000:
"m_590.6"	M 590.6	BOOL	// TL2000:
"m_590.7"	M 590.7	BOOL	// TL2000:
"m_591.0"	M 591.0	BOOL	// TL2000:
"m_591.1"	M 591.1	BOOL	// TL2000:
"m_591.2"	M 591.2	BOOL	// TL2000:
"m_591.3"	M 591.3	BOOL	// TL2000:
"m_591.4"	M 591.4	BOOL	// TL2000:
"m_591.5"	M 591.5	BOOL	// TL2000:
"m_591.6"	M 591.6	BOOL	// TL2000:
"m_591.7"	M 591.7	BOOL	// TL2000:
"m_592.0"	M 592.0	BOOL	// TL2000:
"m_592.1"	M 592.1	BOOL	// TL2000:
"m_592.2"	M 592.2	BOOL	// TL2000:
"m_592.3"	M 592.3	BOOL	// TL2000:
"m_592.4"	M 592.4	BOOL	// TL2000:
"m_592.5"	M 592.5	BOOL	// TL2000:
"m_592.6"	M 592.6	BOOL	// TL2000:
"m_592.7"	M 592.7	BOOL	// TL2000:
"m_593.0"	M 593.0	BOOL	// TL2000:
"m_593.1"	M 593.1	BOOL	// TL2000:
"m_593.2"	M 593.2	BOOL	// TL2000:
"m_593.3"	M 593.3	BOOL	// TL2000:
"m_593.4"	M 593.4	BOOL	// TL2000:
"m_593.5"	M 593.5	BOOL	// TL2000:
"m_593.6"	M 593.6	BOOL	// TL2000:
"m_593.7"	M 593.7	BOOL	// TL2000:
"m_594.0"	M 594.0	BOOL	// TL2000:
"m_594.1"	M 594.1	BOOL	// TL2000:
"m_594.2"	M 594.2	BOOL	// TL2000:
"m_594.3"	M 594.3	BOOL	// TL2000:
"m_594.4"	M 594.4	BOOL	// TL2000:
"m_594.5"	M 594.5	BOOL	// TL2000:
"m_594.6"	M 594.6	BOOL	// TL2000:
"m_594.7"	M 594.7	BOOL	// TL2000:
"M_MTaster_Ueberw_aktiv"	M 595.0	BOOL	// TL2000:
"M_MSST_nicht_bereit"	M 595.1	BOOL	// Messtaster in Messzyklus oder Überwachung und nicht bereit
"M_MTaster_Cycle_aktiv"	M 595.2	BOOL	// TL2000:
"M_Neu_Trigg_MSST"	M 595.3	BOOL	// TL2000:
"m_595.4"	M 595.4	BOOL	// TL2000:
"m_595.5"	M 595.5	BOOL	// TL2000:
"m_595.6"	M 595.6	BOOL	// TL2000:
"m_595.7"	M 595.7	BOOL	// TL2000:
"M_Einricht_Sperr_Ax1"	M 596.0	BOOL	// TL2000:
"M_Einricht_Sperr_Ax2"	M 596.1	BOOL	// TL2000:
"M_Einricht_Sperr_Ax3"	M 596.2	BOOL	// TL2000:
"M_Einricht_Sperr_Ax4"	M 596.3	BOOL	// TL2000:
"M_Einricht_Sperr_Ax5"	M 596.4	BOOL	// TL2000:
"m_596.5"	M 596.5	BOOL	// TL2000:
"m_596.6"	M 596.6	BOOL	// TL2000:
"m_596.7"	M 596.7	BOOL	// TL2000:
"m_597.0"	M 597.0	BOOL	// TL2000:
"m_597.1"	M 597.1	BOOL	// TL2000:
"m_597.2"	M 597.2	BOOL	// TL2000:
"m_597.3"	M 597.3	BOOL	// TL2000:
"m_597.4"	M 597.4	BOOL	// TL2000:
"m_597.5"	M 597.5	BOOL	// TL2000:
"m_597.6"	M 597.6	BOOL	// TL2000:
"m_597.7"	M 597.7	BOOL	// TL2000:
"m_598.0"	M 598.0	BOOL	// TL2000:
"m_598.1"	M 598.1	BOOL	// TL2000:
"m_598.2"	M 598.2	BOOL	// TL2000:
"m_598.3"	M 598.3	BOOL	// TL2000:
"m_598.4"	M 598.4	BOOL	// TL2000:
"m_598.5"	M 598.5	BOOL	// TL2000:
"m_598.6"	M 598.6	BOOL	// TL2000:
"m_598.7"	M 598.7	BOOL	// TL2000:
"m_599.0"	M 599.0	BOOL	// TL2000:
"m_599.1"	M 599.1	BOOL	// TL2000:
"m_599.2"	M 599.2	BOOL	// TL2000:
"m_599.3"	M 599.3	BOOL	// TL2000:
"m_599.4"	M 599.4	BOOL	// TL2000:
"m_599.5"	M 599.5	BOOL	// TL2000:
"m_599.6"	M 599.6	BOOL	// TL2000:
"m_599.7"	M 599.7	BOOL	// TL2000:
"M_FP_HAUPTPROGRAMM_ENDE"	M 600.0	BOOL	// Hauptprogramm Ende Flanke Positiv
"M_Bremsen_Zu_Verz_ESR"	M 600.5	BOOL	// DM_ESR: Verzögertes abschalten der Bremsen um Rückzug zu gewährleisten
"M_GE_Spindellast_aktiv"	M 601.0	BOOL	// General Electric Spezifikation: Spindellastüberwachung ist aktiv
"M_GE_Spindeldrehzahl_akt"	M 601.1	BOOL	// General Electric Spezifikation: Spindeldrehzahlüberwachung ist aktiv
"M_GE_KMTL_Durchfl_aktiv"	M 601.2	BOOL	// General Electric Spezifikation: Kühlmitteldurchflussüberwachung ist aktiv
"M_GE_OMAT_Vorschubsperre"	M 601.3	BOOL	// General Electric Spezifikation: OMATIVE ACM Vorschubsperre ausgelöst
"M_FP_GE_OMAT_ALARM"	M 601.4	BOOL	// General Electric Spezifikation: OMATIVE ACM Flanke Alarm ausgelöst
"M_GE_VS_OVR_gesperrt"	M 601.5	BOOL	// General Electric Spezifikation: Vorschub Override wird durch Omative gesperrt
"M_GE_SPI_OVR_gesperrt"	M 601.6	BOOL	// General Electric Spezifikation: Spindeloverride wird von Omative gesperrt
"M_FD_DM_TURN_AKTIV"	M 601.7	BOOL	// Zyklus DM_TURN ist aktiv
"O_ROBOT_ADR_W0"	M 602.0	BOOL	// Data-Bit 0
"O_ROBOT_ADR_W1"	M 602.1	BOOL	// Data-Bit 1
"O_ROBOT_ADR_W2"	M 602.2	BOOL	// Data-Bit 2
"O_ROBOT_ADR_W3"	M 602.3	BOOL	// Data-Bit 3
"O_ROBOT_ADR_W4"	M 602.4	BOOL	// Data-Bit 4
"O_ROBOT_ADR_W5"	M 602.5	BOOL	// Data-Bit 5
"O_ROBOT_ADR_W6"	M 602.6	BOOL	// Data-Bit 6
"O_ROBOT_ADR_W7"	M 602.7	BOOL	// Data-Bit 7
"O_ROBOT_ADR_W8"	M 603.0	BOOL	// Data-Bit 8
"O_ROBOT_ADR_C0"	M 603.1	BOOL	// Data-Bit 0 C
"O_ROBOT_ADR_C1"	M 603.2	BOOL	// Data-Bit 1 C
"O_ROBOT_ADR_PARITY"	M 603.3	BOOL	// Parity-Bit
"M_ROBOT_DATA"	M 607.0	BOOL
"M_SERIELL_ADRESS_AKTIV"	M 608.0	BOOL	// Adressübertragung an Handlingsystem aktiv
"M_HANDLINGSYSTEM_AKTIV"	M 608.1	BOOL	// Werkstückwechsel durch Handlingsystem aktiv
"M_FN_ROBOT_CLOCK"	M 608.3	BOOL
"M_CHECK_DATA_IN"	M 608.4	BOOL
"M_ROBOT_SYNC"	M 608.5	BOOL
"M_POS_TAKT"	M 608.6	BOOL
"M_NEG_TAKT"	M 608.7	BOOL
"M_ROBOT_DOOR_OPEN"	M 609.0	BOOL	// Beladetür Handlingsystem öffnen
"M_ROBOT_DOOR_CLOSE"	M 609.1	BOOL	// Beladetür Handlingsystem schliessen
"M_FP_MSSTstReset"	M 609.2	BOOL	// Positive Flanke Resettaste
"M_FP_RPC_NC-START"	M 609.3	BOOL	// Positiveflanke NC_Start durch Siemens RPC
"M_FP_8_ter_OB1_Zyklus"	M 609.4	BOOL
"M_NC_START_RPC_3R"	M 609.5	BOOL	// NC-Start durch Handlingsystem 3R
"M_NC_STOP_RPC_3R"	M 609.6	BOOL	// NC-Stop durch Handlingsystem 3R
"M_RESET_RPC_3R"	M 609.7	BOOL	// Reset durch Handlingsystem 3R
"M_ROBOT_DATA_IN"	M 610.7	BOOL	// Serielles Adressbit der zurückgesandten Adresse des Handlingsystem 3R
"M_VMS_MESSAGE_WINDOW"	M 615.6	BOOL	// Spindelüberwachung Merker für Meldefenster
"M_FP_VMS_CRASH"	M 615.7	BOOL	// Spindelüberwachung Flankenmerker Stosserkennung
"M_FN_WZB_Anf_Lesen"	M 620.0	BOOL
"M_IMP_WZB_Messung"	M 620.1	BOOL
"O_AL_Messdose_abblasen"	M 620.2	BOOL	// M-AUSGANG: Blasluft Reinigung Werkzeugvermessung |
"Mx_FP_HPT_ENDE"	M 620.3	BOOL	// Positive Flanke Hauptprogramm Ende -> Kabinentür entriegeln
"m_pwgf_PwRset"	M 621.0	BOOL	// Pw Grundstlg.fahren:Pw.Reset
"m_pwgf_Pwh"	M 621.1	BOOL	// Pw Grundstlg.fahren:PalWechsler heben
"m_pwgf_Pws"	M 621.2	BOOL	// Pw Grundstlg.fahren:PalWechsler senken
"m_pwgf_Mdkh"	M 621.3	BOOL	// Pw Grundstlg.fahren:Medienkupplung kuppeln
"m_pwgf_Mdks"	M 621.4	BOOL	// Pw Grundstlg.fahren:Medienkupplung entkuppeln
"m_pwgf_PArKlLoe"	M 621.5	BOOL	// Pw Grundstlg.fahren:Palette ArbRaum entklemmen
"m_pwgf_PArKlemm"	M 621.6	BOOL	// Pw Grundstlg.fahren:Palette ArbRaum klemmen
"m_pwgf_Pwd0"	M 621.7	BOOL	// Pw Grundstlg.fahren:PalWechsler drehen -> 0°
"m_pwgf_Pwd180"	M 622.0	BOOL	// Pw Grundstlg.fahren:PalWechsler drehen -> 180°
"m_pwgf_PKtrPnE"	M 622.1	BOOL	// Pw Grundstlg.fahren:Pal.Anwesenheitskontrolle im ArbRaum:Luft Ein
"m_pwgf_PKtrPnA"	M 622.2	BOOL	// Pw Grundstlg.fahren:Pal.Anwesenheitskontrolle im ArbRaum:Luft Aus
"m_pwgf_KmPE"	M 622.3	BOOL	// Pw Grundstlg.fahren:KmPumpe Tischspülung ein
"m_pwgf_KmPA"	M 622.4	BOOL	// Pw Grundstlg.fahren:KmPumpe Tischspülung aus
"m_pwgf_PRpKlemm"	M 622.5	BOOL	// Pw Grundstlg.fahren:Palette Rüstplatz klemmen
"m_pwgf_CRqPwPos"	M 622.6	BOOL	// Pw Grundstlg.fahren:C-Achse Pw-Pos.anfahren
"m_pwgf_TiAxRqDp"	M 622.7	BOOL	// Pw Grundstlg.fahren:Tischachse freifahren zur Drehpos(bei SchwenkRt
"m_pwgf_TiAxRqPw"	M 623.0	BOOL	// Pw Grundstlg.fahren:Tischachse fahren zur PalWechsPos.
"m_pwgf_StpAsup2"	M 623.1	BOOL	// Pw Grundstlg.fahren: Halt ASUP_MACHINE Nr.2
"m_pwgf_KmVE"	M 623.2	BOOL	// Pw Grundstlg.fahren:KmVentil Tischspülung ein
"m_pwgf_KmVA"	M 623.3	BOOL	// Pw Grundstlg.fahren:KmVentil Tischspülung aus
"m_pwgf_PKtrNPnE"	M 623.4	BOOL	// Pw Grundstlg.fahren::Pal.Anwesenheitsktrl.im ArbRaum:neg.Ventil Luft Ein
"m_pwgf_PKtrNPnA"	M 623.5	BOOL	// Pw Grundstlg.fahren::Pal.Anwesenheitsktrl.im ArbRaum:neg.Ventil Luft Aus
"m_pwgf_MdkhSp"	M 623.6	BOOL	// Pw Grundstlg.fahren:Medienkupplung ankuppeln nicht FD
"m_pwgf_RPMdkhSp"	M 623.7	BOOL	// Pw Grundstlg.fahren:Rüstplatz Medienkupplung kuppeln
"m_pwfr_0Gad_Pos"	M 624.0	BOOL	// Keine Vorschubfreigabe der Tischachse während des PW
"m_pw_Tisch_0Grad"	M 624.1	BOOL	// PW Tisch-Achse auf 0 Grad position
"m_reload_move"	M 628.0	BOOL	// Wz.umsort:aus Wizzard: Werkzeuge umsortieren mit Bewegung
"m_StrtRld_move"	M 628.1	BOOL	// Wz.umsort:Start Wz.umsetzen mit Bewegung (reales Umsetzen)
"m_QuRld_nomove"	M 628.2	BOOL	// Wz.umsort:Umsetzen ohne Bewegung fertig (Quittierung)
"m_QuRld_move"	M 628.3	BOOL	// Wz.umsort:Umsetzen mit Bewegung fertig (Quittierung)
"m_TmTBefSr0"	M 628.4	BOOL	// Wz.umsort:SrKette TM_T_Befehl kein Sr.gesetzt, Sr0
"m_RsTm_reload"	M 628.5	BOOL	// Wz.umsort:Reset Wzw FbTM_T_Befehl wegen Wz.physik.umsortieren
"m_RsReload"	M 628.6	BOOL	// Wz.umsort:Reset SS Reloading über FC8
"m628.7"	M 628.7	BOOL	// Wz.umsort:
"m629.0"	M 629.0	BOOL	// Wz.umsort:
"m629.1"	M 629.1	BOOL	// Wz.umsort:
"m629.2"	M 629.2	BOOL	// Wz.umsort:
"m629.3"	M 629.3	BOOL	// Wz.umsort:
"m629.4"	M 629.4	BOOL	// Wz.umsort:
"m629.5"	M 629.5	BOOL	// Wz.umsort:
"m629.6"	M 629.6	BOOL	// Wz.umsort:
"m629.7"	M 629.7	BOOL	// Wz.umsort:
"m630.0"	M 630.0	BOOL	// Wz.umsort:
"m630.1"	M 630.1	BOOL	// Wz.umsort:
"m630.2"	M 630.2	BOOL	// Wz.umsort:
"m630.3"	M 630.3	BOOL	// Wz.umsort:
"m630.4"	M 630.4	BOOL	// Wz.umsort:
"m630.5"	M 630.5	BOOL	// Wz.umsort:
"m630.6"	M 630.6	BOOL	// Wz.umsort:
"m630.7"	M 630.7	BOOL	// Wz.umsort:
"m631.0"	M 631.0	BOOL	// Wz.umsort:
"m631.1"	M 631.1	BOOL	// Wz.umsort:
"m631.2"	M 631.2	BOOL	// Wz.umsort:
"m631.3"	M 631.3	BOOL	// Wz.umsort:
"m631.4"	M 631.4	BOOL	// Wz.umsort:
"m631.5"	M 631.5	BOOL	// Wz.umsort:
"m631.6"	M 631.6	BOOL	// Wz.umsort:
"m631.7"	M 631.7	BOOL	// Wz.umsort:
"M_FP_NC_START_RPC_3R"	M 632.0	BOOL
"M_FP_NC_STOP_RPC_3R"	M 632.1	BOOL
"M_FP_RESET_RPC_3R"	M 632.2	BOOL
"M_IMP_MSST_RESET"	M 632.3	BOOL
"M_IMP_NC_STOP_MSST"	M 632.4	BOOL
"M_FP_MSST_RESET"	M 632.5	BOOL
"M_FP_NC_STOP_MSST"	M 632.6	BOOL
"M_Teilung_neu"	M 633.0	BOOL
"M_PARITY_BIT"	M 633.1	BOOL
"M_SAFETY_SBH_AKTIV"	M 633.2	BOOL	// Safety SBH aktiv --> Freigabe Arbeitsraumtüren entriegeln
"I_WA_ENABLE_DOOR_OPEN"	M 633.3	BOOL	// Freigabe Kabinentüre entriegeln
"M_ROBOT_FAHREN_AUF_WEPOS"	M 633.4	BOOL	// Rettung Achsen auf Wechselposition fahren
"M_ROBOT_FAHREN_AUF_SPPOS"	M 633.5	BOOL	// Rettung Achsen auf Spülposition fahren
"M_FP_ASUP_WEPOS"	M 633.6	BOOL
"M_FP_ASUP_SPPOS"	M 633.7	BOOL
"M_AUF_WE_POS"	M 634.0	BOOL	// Achsen auf Wechselposition für Roboter
"M_AUF_SP_POS"	M 634.1	BOOL	// Achsen auf Spülposition für Roboter
"M_Start_PW_Schrittkette"	M 634.2	BOOL	// Schrittkette für PW-Ablauf starten
"I_TC_MAGAZINPOS"	M 634.3	BOOL
"I_TC_SPIPOS"	M 634.4	BOOL
"O_TC_MAGAZINPOS"	M 634.5	BOOL
"O_TC_SPIPOS"	M 634.6	BOOL
"I_U_AXIS_SWITCH_PLUS"	M 636.0	BOOL	// M-EINGANG: U-Achse Mapal MAX-Endschalter (Hardware) erreicht
"I_U_AXIS_SWITCH_MINUS"	M 636.1	BOOL	// M-EINGANG: U-Achse Mapal MIN-Endschalter (Hardware) erreicht
"I_U_AXIS_READY"	M 636.2	BOOL	// M-EINGANG: U-Achse Mapal betriebsbereit
"I_U_AXIS_REF_SIGNAL"	M 636.3	BOOL	// M-EINGANG: U-Achse Mapal Referenzsignal
"I_U_AXIS_ERROR"	M 636.4	BOOL	// M-EINGANG: U-Achse Mapal interner Fehler
"I_U_AXIS_OK"	M 636.5	BOOL	// M-EINGANG: U-Achse Mapal in Ordnung
"I_U_AXIS_CONTROL_READY"	M 636.6	BOOL	// M-EINGANG: U-Achse Mapal Rechner bereit
"I_U_AX_SWITCH_SOFTW_MIN"	M 636.7	BOOL	// M-EINGANG: U-Achse Mapal MIN-Endschalter (Software) erreicht
"I_U_AX_SWITCH_SOFTW_MAX"	M 637.0	BOOL	// M-EINGANG: U-Achse Mapal MAX-Endschalter (Software) erreicht
"I_U_AXIS_RESERVE_1"	M 637.1	BOOL	// M-EINGANG: U-Achse Mapal Reserve 1
"I_U_AXIS_RESERVE_2"	M 637.2	BOOL	// M-EINGANG: U-Achse Mapal Reserve 2
"I_U_AXIS_RESERVE_3"	M 637.3	BOOL	// M-EINGANG: U-Achse Mapal Reserve 3
"I_U_AXIS_RESERVE_4"	M 637.4	BOOL	// M-EINGANG: U-Achse Mapal Reserve 4
"I_U_AXIS_RESERVE_5"	M 637.5	BOOL	// M-EINGANG: U-Achse Mapal Reserve 5
"O_U_AXIS_TOOL_ON"	M 637.6	BOOL	// M-AUSGANG: U-Achse Mapal Werkzeug ist angekoppelt, Betriebsbereitschaft
"O_U_AXIS_RESERVE"	M 637.7	BOOL	// M-AUSGANG: U-Achse Mapal Reserve
"O_U_AXIS_ENABLE_ROTOR"	M 638.0	BOOL	// M-AUSGANG: U-Achse Mapal Freigabe Rotor
"O_U_AXIS_QUIT"	M 638.1	BOOL	// M-AUSGANG: U-Achse Mapal Rücksetzen, Fehlerquittierung, Reset
"O_U_AXIS_PROFILE_ACTIV"	M 638.2	BOOL	// M-AUSGANG: U-Achse Mapal Profil aktivieren
"O_U_AXIS_EAT_LAT"	M 638.3	BOOL	// M-AUSGANG: U-Achse Mapal Auswahl EAT oder LAT (Exzenter oder Linear) 1--> LAT
"O_U_AXIS_PROFILE_BIT_0"	M 638.4	BOOL	// M-AUSGANG: U-Achse Mapal Profil Bit 0
"O_U_AXIS_PROFILE_BIT_1"	M 638.5	BOOL	// M-AUSGANG: U-Achse Mapal Profil Bit 1
"O_U_AXIS_PROFILE_BIT_2"	M 638.6	BOOL	// M-AUSGANG: U-Achse Mapal Profil Bit 2
"O_U_AXIS_PROFILE_BIT_3"	M 638.7	BOOL	// M-AUSGANG: U-Achse Mapal Profil Bit 3
"O_U_AXIS_PROFILE_BIT_4"	M 639.0	BOOL	// M-AUSGANG: U-Achse Mapal Profil Bit 4
"O_U_AXIS_PROFILE_BIT_5"	M 639.1	BOOL	// M-AUSGANG: U-Achse Mapal Profil Bit 5
"M_FP_U_AXIS_SWITCH_MAX"	M 640.0	BOOL	// Flankenmerker U-Achse Mapal Endschalter MAX
"M_FP_U_AXIS_SWITCH_MIN"	M 640.1	BOOL	// Flankenmerker U-Achse Mapal Endschalter MIN
"O_WA_REQUEST_DOOR_UNLOC"	M 663.0	BOOL	// Anforderung Kabinentür entriegeln
"I_CU_SAVETY_EMSTP_EN"	M 670.0	BOOL
"I_CU_SAVETYUNIT_CAB_EN"	M 670.1	BOOL
"O_VMS_MSG_FPRINT_START"	M 670.2	BOOL	// IFM-Vibrationsüberwachung Fingerprint-Messung starten
"I_VMS_BEARING_ERROR"	M 670.3	BOOL
"I_VMS_BEARING_WAR"	M 670.4	BOOL
"I_VMS_CRASH"	M 670.5	BOOL
"I_VMS_MEASURING_BEA_RDY"	M 670.6	BOOL
"I_VMS_UNBALANCE_ERROR"	M 670.7	BOOL
"I_VMS_UNBALANCE_WAR"	M 671.0	BOOL
"I_VMS_VIBRATION_FAULT_D"	M 671.1	BOOL
"O_VMS_MSG_BEA_START"	M 671.2	BOOL
"O_RELEASEUNI_GET_TOOL"	M 671.3	BOOL	// Ausrückstation Hub Richtung Werkzeugkegel
"I_RELEASEUNI_GET_TOOL"	M 671.4	BOOL	// Ausrückstation Position Werkzeugkegel
"O_RELEASEUNI_RELEASE_T"	M 671.5	BOOL	// Ausrückstation Hub in Grundstellung
"I_RELEASEUNI_RELEASE_T"	M 671.6	BOOL	// Ausrückstation Position Grundstellung
"O_RELEASEUNI_TRANSPOS"	M 671.7	BOOL	// Ausrückstation Hub Richtung Übergabeposition
"I_RELEASEUNI_TRANSPOS"	M 672.0	BOOL	// Ausrückstation Position Übergabeposition
"O_RELEASEUNI_MAGAZINPOS"	M 672.1	BOOL	// Ausrückstation Richtung Magazinposition
"I_RELEASEUNI_MAGAZINPOS"	M 672.2	BOOL	// Ausrückstation Position Magazinposition
"O_RELU_MAG_TOOL_UNLOC"	M 672.3	BOOL	// Ausrückstation WZ Greifer entriegeln
"I_RELU_MAG_TOOL_UNLKD"	M 672.4	BOOL	// Ausrückstation Werkzeug im Greifer gelöst
"I_RELU_MAG_TOOL_LKD"	M 672.5	BOOL	// Ausrückstation Werkzeug im Greifer gespannt
"I_RELU_MAG_PIN_LKD"	M 672.6	BOOL	// Ausrückstation Verriegelungspin Magazinplatz verriegelt
"I_RELEASEUNI_MAG_OCC"	M 672.7	BOOL	// Ausrückstation Magazinplatz belegt
"O_RELU_TST_TOOL_UNLOC"	M 673.0	BOOL	// Ausrückstation WZ-Pin Magazinplatz entriegeln
"I_RELU_TST_TOOL_UNLKD"	M 673.1	BOOL	// Ausrückstation Kettenverriegelungszylinder ausgefahren
"I_RELEASEUNI_TST_OCC"	M 673.2	BOOL	// Ausrückstation Übergabeplatz belegt
"I_RELU_TST_TOOL_LKD"	M 673.3	BOOL	// Ausrückstation Kettenverriegelungszylinder eingefahren
"O_RELU_TOOL_C_BL_AI"	M 673.4	BOOL	// Ausrückstation Blasluft Kegel- und Sensorreinigung
"Start_ASUP_Machine_Nr.8"	M 688.1	BOOL	// ASUP-fc201 8 Roboter Rettung
"I_SPI_WZ_SPA_UEBERW_ZUG"	M 704.0	BOOL	// Überwachung Löseeinheit Analog Spanner
"M_WZ_SPA_gesp_Analog"	M 704.1	BOOL	// Merker Analog Spanner gespannt
"M_WZ_SPA_geloe_Analog"	M 704.2	BOOL	// Merker Analog Spanner gelöst
"M_WZ_equal_alt_neu"	M 704.7	BOOL	// Werkzeugtyp altes WZ ist gleich neues WZ
"M_FEHL_ÜBERW"	M 705.0	BOOL	// Fehlerüberwachung MMS Fa.Vogel
"M_MinMg_Schmier_Aktiv"	M 705.1	BOOL	// Minimalmengenschmierung Fa. Vogel
"FP_Glaet_aktiv"	M 706.0	BOOL	// Impuls Glaettung aktiv
"FP_Glaet_aktiv1"	M 706.1	BOOL
"MX_ACESSS_LEVEL_1"	M 707.0	BOOL	// Schlüsselschalter 0
"MX_ACESSS_LEVEL_2"	M 707.1	BOOL	// Schlüsselschalter 1
"MX_ACESSS_LEVEL_3"	M 707.2	BOOL	// Schlüsselschalter 2
"MX_ACESSS_LEVEL_4"	M 707.3	BOOL	// Schlüsselschalter 3
"MX_ACESSS_LEVEL_5"	M 707.4	BOOL	// Anwender - Customer
"MX_ACESSS_LEVEL_6"	M 707.5	BOOL	// Service - Evening/Hersteller - Auduser
"MX_ACESSS_LEVEL_7"	M 707.6	BOOL	// System
"MX_ACESSS_LEVEL_8"	M 707.7	BOOL
"I_GEN_OM_BIT_0"	M 708.0	BOOL	// Smartkey - Betriebsart BA1 - BA4 / Meldung 0-3
"I_GEN_OM_BIT_1"	M 708.1	BOOL	// Smartkey - Betriebsart BA1 - BA4 / Meldung 0-3
"I_GEN_OM_BIT_2"	M 708.2	BOOL	// Smartkey - Berechtigung / Meldung
"I_GEN_OM_BIT_3"	M 708.3	BOOL	// Smartkey - Anwahl / Meldung
"I_GEN_OM_BIT_4"	M 708.4	BOOL	// Reserve
"I_GEN_OM_BIT_5"	M 708.5	BOOL	// Reserve
"I_GEN_OM_BIT_6"	M 708.6	BOOL	// Reserve
"I_GEN_OM_BIT_7"	M 708.7	BOOL	// Reserve
"I_GEN_OM_SERVICE_ACTIVE"	M 709.0	BOOL	// Smartkey - Service-Betriebsart aktiv
"Mx_FP_20MinPasswrt_rueck"	M 709.1	BOOL
"I_GEN_PLC_DATA_SEL"	M 709.2	BOOL	// Eingabe der PLC Daten wurde freigegeben
"M_SPI_Load_Alert"	M 724.0	BOOL	// Omative ACM: Spindelleistungüberwachung hat ausgelöst
"M_SPI_Speed_Alert"	M 724.1	BOOL	// Omative ACM: Spindeldrehzahlüberwachung hat ausgelöst
"mx_FP_PW_aktiv"	M 734.0	BOOL	// Positive Flanke PW aktiv
"mx_FP_PW_Time_Hub_senk"	M 734.1	BOOL
"mx_FP_MPL_Abfra_Ventil"	M 734.2	BOOL	// Ventil Luftstrom Palette aktivieren
"mx_FP_deakti_Ventil_Abfr"	M 734.3	BOOL	// Deaktivierung Ventil Luftstrom Palette nach der Pruefung MPL
"mx_time_aktiv_hub_senk"	M 734.4	BOOL	// Hub senken aktiv bis PW in Mittelstellung
"mx_FP_Time_Zwis"	M 734.5	BOOL	// Zeit PW-senken in Zwischenspeicher schreiben
"mx_MPL_Abfr_2_Hubbew"	M 734.6	BOOL	// Palettenkontrolle wurde nicht korrekt ausgeführt 2 Hubbewegung
"mx_MPL_Abfr_3_Hubbew"	M 734.7	BOOL	// Palettenkontrolle wurde nicht korrekt ausgeführt 3 Hubbewegung
"M_BrushClean_Signal_NOK"	M 800.0	BOOL	// Kegelreinigung Stoerung Paarueberwachung
"M_BrushClean_Strg_AST"	M 800.1	BOOL	// Kegelreinigung Stoerung Laufzeit Arbeitsstellung
"M_BrushClean_Strg_GST"	M 800.2	BOOL	// Kegelreinigung Stoerung Laufzeit Grundstellung
"MX_SKEY_IDENT_SENDEN"	M 814.0	BOOL	// Start zum Senden der Smartkey Identnummer
"MX_SKEY_TOGGLE_TAG"	M 814.1	BOOL
"M_WZ_Sperren_REQUEST"	M 859.0	BOOL
"M_WZ_Sperren_ERROR"	M 859.1	BOOL
"M_WZ_Sperren_DONE"	M 859.2	BOOL
"WZB_2_MESSUNG_ABLEGEN"	M 888.0	BOOL	// WZW VK: WZ-Bruch Start 2 Messung durch Ablauf Ablegen
"WZB_2_MESSUNG_FERTIG"	M 888.1	BOOL	// WZW VK: WZ-Bruch 2 Messung ist fertig
"WZB_PARKPOSITION_FP"	M 888.2	BOOL	// WZW VK: WZ-Bruch in Parkposition Flanke positiv
"WZB_MESSUNG_AUSGEFUEHRT"	M 888.3	BOOL	// WZW VK: WZ-Bruch Messung wurde ausgeführt
"M_WZW_MAG_ABBR_POS"	M 888.4	BOOL	// WZW: Magazinachse Abbruch Positionierung während der Bewegung
"M_WZW_MAG_START_N_RESET"	M 888.5	BOOL	// WZW: Start Magazinpositionierung nach Reset
"M_WZW_MAG_IN_UEBERGABE"	M 888.6	BOOL	// WZW: MAgazin in Übergabestellung
"M_CAMPSTAND_AKTIV"	M 888.7	BOOL	// Campstand aktiv ( Merker kann 0/1 gesetzt werden für Testzwecke am Campstand)
"M_WZW_QUITT_FEHLENDES_WZ"	M 889.0	BOOL	// WZW: Quittierung fehlendes Werkzeug beladen durch Beladeklappe zu
"M_WZW_QUITT_FEHL_WZ_FP"	M 889.1	BOOL	// WZW: Quittierung fehlendes Werkzeug beladen durch Beladeklappe zu Flanke positiv
"WZB_FRUEHSTART_AUSLOESEN"	M 889.2	BOOL	// WZW VK: WZ-Bruch Frühstart auslösen
"M_FP_TE_MASCHINE_EIN"	M 889.7	BOOL
"M_RPT_SIMULATION_ZU"	M 900.0	BOOL	// Simulations-Kommando RPL-Tür zu
"M_RPT_SIMULATION_AUF"	M 900.1	BOOL	// Simulations-Kommando RPL-Tür auf
"M_RPT_Simulation"	M 900.7	BOOL	// Rp-Tür Si mulation ist aktiv
"I_AL_Sicherung_24V_OK"	M 999.0	BOOL	// M-EINGANG: Diagnose Sicherung 24V
"I_AL_SICHERUNG_230V_OK"	M 999.1	BOOL	// M-EINGANG: Diagnose Sicherung 230V
"O_SO_WFK_UMSCH_KM"	M 999.7	BOOL	// M-AUSGANG: Wiegenfräskopf Kühlmittel Umschaltung
"Error_FB_SIEM_PUT_GUDs"	M 1000.0	BOOL	// Error-Meldung von Baustein FB_SIEM_PUT beim Ablegen der GUDs
"Done_FB_SIEM_PUT_GUDs"	M 1000.1	BOOL	// Done-Meldung von Baustein FB_SIEM_PUT beim Ablegen der GUDs
"O_ROBOT_CLOCK"	M 1007.0	BOOL	// Ueberwachung Takt
"O_ROBOT_COP1"	M 1007.1	BOOL	// Freigabe Spannfutter
"O_ROBOT_DATA"	M 1007.2	BOOL	// Adresse Uebertragung
"O_ROBOT_DOOR_CLOSE"	M 1007.3	BOOL	// Hubtuere Werkstueckmagazin schliessen
"O_ROBOT_DOOR_OPEN"	M 1007.4	BOOL	// Hubtuere Werkstueckmagazin oeffnen
"O_ROBOT_SYNC"	M 1007.6	BOOL
"O_ROBOT_TCP1"	M 1007.7	BOOL
"I_AL_BA_SERVICE_AKTIV"	M 1008.0	BOOL
"I_ROBOT_AUTO"	M 1008.1	BOOL	// Handlingsystem in Automatikbetrieb
"I_ROBOT_CHUCKS_CLOSED"	M 1008.3	BOOL	// Spannfutter gespannt
"I_ROBOT_DATA_IN"	M 1008.4	BOOL	// Adresse Rueckmeldung
"I_ROBOT_DOOR_CLOSED"	M 1008.5	BOOL
"I_ROBOT_DOOR_OPENED"	M 1008.6	BOOL	// Hubtuere Werkstueckmagazin offen
"I_ROBOT_NEG_ERROR"	M 1008.7	BOOL	// Fehler Handlingsystem
"O_SK_VER_schwenken"	M 1009.0	BOOL	// M-AUSGANG: Schwenkfraeskopf senkrecht M54
"O_SK_HOR_schwenken"	M 1009.1	BOOL	// M-AUSGANG: Schwenkfraeskopf waagrecht M53
"O_SK_Klemmung_loesen"	M 1009.2	BOOL	// M-AUSGANG: Schwenkfraeskopf Klemmung loesen
"O_SK_Klemmung_zu"	M 1009.3	BOOL	// M-AUSGANG: Schwenkfraeskopf Klemmung klemmen
"I_ROBOT_ERROR"	M 1009.4	BOOL	// Fehler Handlingsystem 3R
"O_KM_SPUELUNG_GREIFER"	M 1009.5	BOOL
"I_ROBOT_NEUTRAL"	M 1009.6	BOOL	// Grundstellung Handlingsystem
"M_Mel_MAX_Fuell_Kratz"	M 1009.7	BOOL
"I_AL_Vorschubfreigabe"	M 1010.0	BOOL	// M-EINGANG: Vorschubfreigabe X/Y/Z-Achse 4./5.-Achse
"I_AL_EINLESEFREIGABE"	M 1010.1	BOOL	// M-EINGANG: Einlesefreigabe
"I_AL_DISABLE_POWERSAVE"	M 1010.4	BOOL	// M-EINGANG: Freigabe
"I_AL_NEG_MSS_Kuehlung"	M 1010.5	BOOL	// M-EINGANG: Motorschutzschalter Luefter Waermetauscher Kuehlaggregat
"I_SF_Automatik"	M 1011.0	BOOL	// M-EINGANG: Spaenefoerderer Betriebsart Automatik
"I_SF_SCHALTER_RECHTS"	M 1011.1	BOOL	// M-EINGANG: Spaenefoerderer Rechtslauf
"I_LA_dynamisches_Signal"	M 1011.2	BOOL	// M-EINGANG: LA: Laser Signal dynamisch
"I_MAS_NEG_SPANNDRUCK"	M 1011.4	BOOL	// M-EINGANG: Druckschalter Spannvorrichtung geloest
"I_AL_4ACHS_KLE_auf"	M 1011.5	BOOL	// M-EINGANG: Klemmung 4.Achse auf
"I_AL_4ACHS_KLE_geloest"	M 1011.6	BOOL	// M-EINGANG: Klemmung 4.Achse gelöst
"I_AL_4ACHS_KLE_zu"	M 1011.7	BOOL	// M-EINGANG: Klemmung 4.Achse zu
"I_AL_5ACHS_KLE_geloest"	M 1012.0	BOOL	// M-EINGANG: Klemmung 5./11. Achse gelöst
"M_FP_START_FC8"	M 1012.1	BOOL
"I_WM_TAS_Beladung_zu"	M 1012.2	BOOL	// M-EINGANG: Freigabe Magnetverriegelung WZB-geschlossen
"I_WM_Beladung_auf"	M 1012.3	BOOL	// M-EINGANG: Werkzeugbestueckung Fenster geoffnet
"I_WM_1_Eingabeplatz"	M 1012.4	BOOL	// M-EINGANG: Ueberwachung Werkzeugbestueckung Platz 1
"M_FP_FMS_T_ENTL"	M 1012.6	BOOL
"I_WM_Eing_Station"	M 1012.7	BOOL	// M-EINGANG: Umschaltung Werkzeugeingabefunktion
"I_WM_2_Eingabeplatz"	M 1013.2	BOOL	// M-EINGANG: Ueberwachung Werkzeugbestueckung Platz 2
"I_WM_3_Eingabeplatz"	M 1013.3	BOOL	// M-EINGANG: Ueberwachung Werkzeugbestueckung Platz 3
"I_WM_4_Eingabeplatz"	M 1013.4	BOOL	// M-EINGANG: Ueberwachung Werkzeugbestueckung Platz 4
"I_WW_Ablageplatz"	M 1013.5	BOOL	// M-EINGANG: Ueberwachung Ablageplatz Handlingsystem
"I_D_WW_Ablageplatz"	M 1013.6	BOOL	// M-EINGANG: Diagnose Ueberwachung Ablageplatz
"I_WM_TOPF_SPA_OFFEN"	M 1013.7	BOOL	// M-EINGANG: Pneumatikzylinder Werkzeugspanner geoeffnet
"I_WM_TOPF_SPA_ZU_MIT_WZ"	M 1014.0	BOOL	// M-EINGANG: Pneumatikzylinder Werkzeugspanner geschlossen mit Werkzeug
"I_WM_TOPF_SPA_ZU_O_WZ"	M 1014.1	BOOL	// M-EINGANG: Pneumatikzylinder Werkzeugspanner geschlossen ohne Werkzeug
"M_IMP_H20_Quit"	M 1014.6	BOOL
"M_FP_H20_Quit"	M 1014.7	BOOL
"OX_SP_RPL_FREIGABE"	M 1017.6	BOOL	// M-AUSGANG: Freigabe SpannHydraulik Rüstplatz
"OX_RPL_TUER_OEFFNEN"	M 1018.4	BOOL	// M-AUSGANG: Ventil Rüstplatztür öffnen
"OX_RPL_TUER_SCHLIESSEN"	M 1018.5	BOOL	// M-AUSGANG: Ventil Rüstplatztür schließen
"I_PW_RPL_PAL_GEKLEMMT"	M 1019.0	BOOL	// M-EINGANG: Ruestplatz Palettenklemmung geklemmt
"I_PW_RPL_PAL_GELOEST"	M 1019.1	BOOL	// M-EINGANG: Ruestplatz Palettenklemmung geloest
"O_PW_RPL_PAL_KLEMMEN"	M 1019.2	BOOL	// M-AUSGANG: Ruestplatz Palettenklemmung klemmen
"O_PW_RPL_PAL_LOESEN"	M 1019.3	BOOL	// M-AUSGANG: Ruestplatz Palettenklemmung loesen
"O_PW_N_VENTIL_ABFRAGE"	M 1020.0	BOOL	// M-AUSGANG: Druckluft Palettenerkennung
"I_TM_RELEASE"	M 1020.1	BOOL
"I_SST_ENABLE_ROTATE"	M 1021.1	BOOL	// M-EINGANG: Rüstpaltzachse Antriebsfreigabe
"O_AL_4ACHS_KLE_LOESEN"	M 1021.2	BOOL	// M-AUSGANG: 4.Achse Klemmung lösen
"O_PW_SPANNKONEN_ABBLAS"	M 1021.3	BOOL	// M-AUSGANG: Spannkonen abblasen
"Mx_Tisch_geklemmt_Hilfm"	M 1021.4	BOOL	// Hilfsmerker Tischklemmung geklemmt bei Druckerhoehung 180 Ba
"Mx_FP_Tischkl_loes"	M 1021.5	BOOL	// Positive Flanke Tischklemmung loesen
"Mx_FP_1s_Takt"	M 1021.6	BOOL	// Positive Flanke im Sekundentakt
"M_FP_read_pallet_number"	M 1024.0	BOOL
"M_FP_FMS_HYD_INFO"	M 1024.1	BOOL
"I_PC_FIXTURE_EXIST"	M 1040.0	BOOL	// Nullpunktspannsystem Positionsueberwachung Spannvorrichtung
"MX_FIXTURE_ON_APC"	M 1040.1	BOOL	// Nullpunktspannsystem geklemmt
"MX_FIXTURE_RELEASED"	M 1040.2	BOOL	// Nullpunktspannsystem geloest
"I_FMS_FIXTURE_RELEASE"	M 1040.3	BOOL	// Nullpunktspannsystem loesen
"MX_Fixture_Locked"	M 1040.4	BOOL	// Nullpunktspannsystem gespannt
"I_FMS_AUTO_POWER_OFF"	M 1040.5	BOOL	// ME G3-12.x MC INPUT BYTE 1 Bit 3
"I_FMS_OM_DISABLED"	M 1041.0	BOOL	// Schluesselschalter Deaktivierung Uebergabeplatz/ Maschine/Palettenspeichersystem
"O_FMS_OM1_DISABLED"	M 1041.1	BOOL	// Betriebsart Automatik gesperrt Palettenspeichersystem
"Mx_FMS_OM1_DISABLED"	M 1041.2	BOOL	// Freigabe NC_START/ PW_FREIGABE
"I_SF_RECHEN_1_HINTEN"	M 1080.0	BOOL	// Spaenefoerderer -Rechen 1 Hubeinheit hinten
"I_SF_RECHEN_1_VORNE"	M 1080.1	BOOL	// Spaenefoerderer -Rechen 1 Hubeinheit vorn
"I_SF_RECHEN_2_HINTEN"	M 1080.2	BOOL	// Spaenefoerderer -Rechen 2 Hubeinheit hinten
"I_SF_RECHEN_2_VORNE"	M 1080.3	BOOL	// Spaenefoerderer -Rechen 2 Hubeinheit vorn
"I_SF_RECHEN_DRUCKLOS"	M 1080.4	BOOL	// Druckschalter Hauptluft Spaenefoerderer-Rechen
"I_SF_RECHEN_DRUCKLOS_D"	M 1080.5	BOOL	// Diagnose Druckschalter Hauptluft Spaenefoerderer-Rechen
"O_SF_RECHEN_1_VOR"	M 1081.0	BOOL	// Spaenefoerderer- Rechen 1 Hubeinheit vor
"O_SF_RECHEN_1_ZURUECK"	M 1081.1	BOOL	// Spaenefoerderer- Rechen 1 Hubeinheit zurueck
"O_SF_RECHEN_2_VOR"	M 1081.2	BOOL	// Spaenefoerderer- Rechen 2 Hubeinheit vor
"O_SF_RECHEN_2_ZURUECK"	M 1081.3	BOOL	// Spaenefoerderer- Rechen 2 Hubeinheit zurueck
"O_SF_RECHEN_Z_VENTIL"	M 1081.4	BOOL	//  Ventil Hauptluft Spaenefoerderer-Rechen
"Mx_FP_SF_RECH"	M 1081.6	BOOL	// Flankenmerker zuruecksetzen des Zentral-Ventils
"Mx_FP_SF_RECH_AUS"	M 1081.7	BOOL	// Flankenmerker Ruecksetzen der Richtungsventile beim oeffnen der Maschinentuere
"MX_SF_FE_Rechen1"	M 1082.0	BOOL	// Fehlerüberwachung Rechen1
"MX_SF_FE_Rechen2"	M 1082.1	BOOL
"MX_SF_Rechen1_Ein"	M 1082.2	BOOL	// Spaeneförderer-Rechen 1 aktiv
"MX_SF_FB_Rechen1"	M 1082.3	BOOL
"MX_SF_FP1_Rechen1"	M 1082.4	BOOL	// Positive Flanke Rechen 1 vor
"MX_SF_FP2_Rechen1"	M 1082.5	BOOL	// Positive Flanke Rechen 1 zurueck
"MX_TUER_ENTR"	M 1082.6	BOOL	// Positive Flanke Anforderung Tuere oeffnen
"MX_SF_KAB_VERR"	M 1083.0	BOOL	// Positive Flanke Kabienentuer verriegelt
"Mx_RECH_ZUR_TUERAU"	M 1083.1	BOOL
"MX_SF_Rechen2_Ein"	M 1083.2	BOOL
"MX_SF_FB_Rechen2"	M 1083.3	BOOL
"MX_SF_FP1_Rechen2"	M 1083.4	BOOL
"MX_SF_FP2_Rechen2"	M 1083.5	BOOL
"MX_Anf_Tuer_Auf"	M 1083.6	BOOL	// Anforderung Türe auf
"MX_SF_Frg_Tuer_auf"	M 1083.7	BOOL	// Freigabe zum Tür öffnen vom Späneförderer
"M_SF_FP_Rechen1"	M 1084.0	BOOL	// Positive Flanke Rechen 1 Ein
"M_SF_Rechen1_Aktiv"	M 1084.1	BOOL	// Rechen 1 über die Zeit aktiv
"M_SF_FP_Rechen2"	M 1084.2	BOOL	// Positive Flanke Rechen 1 Ein
"M_SF_Rechen2_Aktiv"	M 1084.3	BOOL	// Rechen 2 über die Zeit aktiv
"M_SF_FN2_Rechen1"	M 1084.4	BOOL	// Negative Flanke Rechen1 Zeituberwachung ueberschritten
"M_SF_FN2_Rechen2"	M 1084.5	BOOL	// Negative Flanke Rechen2 Zeituberwachung ueberschritten
"M_FP_PW_AKTIV"	M 1111.1	BOOL
"M_FP_BA_Wechsel_M8_deakt"	M 1111.6	BOOL
"M_FN_Links_drehen"	M 1212.2	BOOL
"M_FN_Rechts_drehen"	M 1212.3	BOOL
"M_PS_RPL_Tuer_zu_GST_fah"	M 1212.4	BOOL	// RPL von PS bei Türe zu in Grundstellung 0-Grad fahren
"M_RPL_in_GST_fahren"	M 1212.5	BOOL
"M_FP_TUER_VORNE_ZU"	M 1212.6	BOOL
"M_SIMULATION_HILFSBIT_0"	M 1888.0	BOOL
"M_SIMULATION_HILFSBIT_1"	M 1888.1	BOOL
"M_SIMULATION_HILFSBIT_2"	M 1888.2	BOOL
"M_SIMULATION_HILFSBIT_3"	M 1888.3	BOOL
"M_SIMULATION_HILFSBIT_4"	M 1888.4	BOOL
"M_SIMULATION_HILFSBIT_5"	M 1888.5	BOOL
"M_SIMULATION_HILFSBIT_6"	M 1888.6	BOOL
"M_SIMULATION_HILFSBIT_7"	M 1888.7	BOOL
"I_SPI_TEMP_RDY"	M 2010.0	BOOL	// M-EINGANG: Temperaturüberwachung Motorspindel (55/65H)
"I_PC_MPL_PALLET_CLPED_D"	M 2010.1	BOOL	// M-EINGANG: Diagnose Palettenklemmung geklemmt  (55/65H)
"I_PC_MPL_PALLET_RELD_D"	M 2010.2	BOOL	// M-EINGANG: Diagnose Palettenklemmung geloest (55/65H)
"I_PC_MPL_OCCUPIED_D"	M 2010.3	BOOL	// M-EINGANG: Diagnose Palette Maschine vorhanden (55/65H)
"I_GEN_HYD_PRESSURE_OK_D"	M 2010.4	BOOL	// M-EINGANG: Diagnose Druckueberwachung Hydraulik (55/65H)
"I_GEN_CAIR_PRE_OK_D"	M 2010.5	BOOL	// M-EINGANG: Diagnose Druckueberwachung Pneumatik (55/65H)
"I_TAB_POSITION_0DEG"	M 2010.6	BOOL	// M-EINGANG: Takttisch in Position 0 Grad
"I_CU_GAP_SCREEN_CL_UPP"	M 2010.7	BOOL	// M-EINGANG:  Kühlmittelanlage Spaltsieb oben
"I_CU_GAP_SCREEN_CL_LOW"	M 2011.0	BOOL	// M-EINGANG:  Kühlmittelanlage Spaltsieb unten
"I_CU_NEG_PRESS_MONITOR"	M 2011.1	BOOL	// M-EINGANG:  Kühlmittelanlage Unterdruck IKZ
"I_TM_PUMP_MPS"	M 2011.2	BOOL	// M-EINGANG:  Motorschutzschalter Hebepumpe Werkzeugmagazin
"I_TM_PUMP_ON"	M 2011.3	BOOL	// M-EINGANG:  Hebepumpe Werkzeugmagazin ein
"I_CU_FLUSH_PIST_SST_ON"	M 2011.4	BOOL	// M-EINGANG:  Spuelpistole Ruestplatz ein
"I_TC_POSITION_BRUSH_CLE"	M 2011.5	BOOL	// M-EINGANG:  Positionsueberwachung Reinigung Werkzeugkegel
"I_TORQ_PROP_FILL_MON"	M 2011.6	BOOL	// M-EINGANG:  Fuellstand Oelbehaelter Drehmomentstuetze
"I_TC_ENABLE"	M 2011.7	BOOL	// M-EINGANG:  Dummy, in PLC  wird "DB_SPL".ISX_TM_DRIVES_EN_CNC abgefragt
"I_PC_ENABLE"	M 2012.0	BOOL	// M-EINGANG: Antriebsfreigabe Palettenwechsler
"I_PC_LIFT_POSITION_4"	M 2012.1	BOOL	// M-EINGANG: Hubeinheit Palettenwechsler Hub schnell
"O_SPI_IMP_DELETE"	M 2030.0	BOOL	// M-AUSGANG: Impuls Hauptantrieb geloescht (55/65H)
"O_INFEED_ENABLE_NCU"	M 2030.1	BOOL	// M-AUSGANG: Ansteuerung NCU: Freigabe Klemme X122.1 SLM bereit (55/65H)
"O_ENABLE_OUT_3_NX_NCU"	M 2030.2	BOOL	// M-AUSGANG: Ansteuerung NCU: Freigabe Klemme X122.2 AUS3 (55/65H)
"O_INFEED_ENABLE_NX"	M 2030.3	BOOL	// M-AUSGANG: Ansteuerung NX: Freigabe Klemme X122.1 Einspeisung ok (55/65H)
"O_CU_GAP_SCREEN_CLEAN"	M 2030.4	BOOL	// M-AUSGANG: Kühlmittelanlage Spaltsieb ein / nach oben  (55/65H)
"O_TM_PUMP"	M 2030.5	BOOL	// M-AUSGANG: Hebepumpe Werkzeugmagazin (55/65H)
"O_CU_FLUSH_PIST_SST_ON"	M 2030.6	BOOL	// M-AUSGANG: Meldung Spuelpistole Ruestplatz ein
"O_TC_ENABLE_BRUSH_CLEAN"	M 2030.7	BOOL	// M-AUSGANG: Freigabe Positionierung Reinigung
"O_TORQ_PROP_CAIR_ON"	M 2031.0	BOOL	// M-AUSGANG: Blasluft Drehmomentstuetze
"O_TC_TL_BRUSH_CLEAN"	M 2031.1	BOOL	// M-AUSGANG: Buerste Reinigung Werkzeugkegel
"O_PC_CLAMP_CONE_BL_O"	M 2031.2	BOOL	// M-AUSGANG: Palettenträger Spannstelle ausblasen
"O_PC_LIFT_FAST_DOWN"	M 2031.3	BOOL	// M-AUSGANG: Hubeinheit Palettenwechsler schnell nach unten
"O_PC_LIFT_FAST_UP"	M 2031.4	BOOL	// M-AUSGANG: Hubeinheit Palettenwechsler schnell nach oben
"M_MAPAL_PROFIL_BIT_24"	M 2040.0	BOOL	// Angewähltes Profil der U-Achse Mapal: Bit von MD_MAPAL_PROFIL
"M_MAPAL_PROFIL_BIT_25"	M 2040.1	BOOL	// Angewähltes Profil der U-Achse Mapal: Bit von MD_MAPAL_PROFIL
"M_MAPAL_PROFIL_BIT_26"	M 2040.2	BOOL	// Angewähltes Profil der U-Achse Mapal: Bit von MD_MAPAL_PROFIL
"M_MAPAL_PROFIL_BIT_27"	M 2040.3	BOOL	// Angewähltes Profil der U-Achse Mapal: Bit von MD_MAPAL_PROFIL
"M_MAPAL_PROFIL_BIT_28"	M 2040.4	BOOL	// Angewähltes Profil der U-Achse Mapal: Bit von MD_MAPAL_PROFIL
"M_MAPAL_PROFIL_BIT_29"	M 2040.5	BOOL	// Angewähltes Profil der U-Achse Mapal: Bit von MD_MAPAL_PROFIL
"M_MAPAL_PROFIL_BIT_30"	M 2040.6	BOOL	// Angewähltes Profil der U-Achse Mapal: Bit von MD_MAPAL_PROFIL
"M_MAPAL_PROFIL_BIT_31"	M 2040.7	BOOL	// Angewähltes Profil der U-Achse Mapal: Bit von MD_MAPAL_PROFIL
"M_MAPAL_PROFIL_BIT_16"	M 2041.0	BOOL	// Angewähltes Profil der U-Achse Mapal: Bit von MD_MAPAL_PROFIL
"M_MAPAL_PROFIL_BIT_17"	M 2041.1	BOOL	// Angewähltes Profil der U-Achse Mapal: Bit von MD_MAPAL_PROFIL
"M_MAPAL_PROFIL_BIT_18"	M 2041.2	BOOL	// Angewähltes Profil der U-Achse Mapal: Bit von MD_MAPAL_PROFIL
"M_MAPAL_PROFIL_BIT_19"	M 2041.3	BOOL	// Angewähltes Profil der U-Achse Mapal: Bit von MD_MAPAL_PROFIL
"M_MAPAL_PROFIL_BIT_20"	M 2041.4	BOOL	// Angewähltes Profil der U-Achse Mapal: Bit von MD_MAPAL_PROFIL
"M_MAPAL_PROFIL_BIT_21"	M 2041.5	BOOL	// Angewähltes Profil der U-Achse Mapal: Bit von MD_MAPAL_PROFIL
"M_MAPAL_PROFIL_BIT_22"	M 2041.6	BOOL	// Angewähltes Profil der U-Achse Mapal: Bit von MD_MAPAL_PROFIL
"M_MAPAL_PROFIL_BIT_23"	M 2041.7	BOOL	// Angewähltes Profil der U-Achse Mapal: Bit von MD_MAPAL_PROFIL
"M_MAPAL_PROFIL_BIT_08"	M 2042.0	BOOL	// Angewähltes Profil der U-Achse Mapal: Bit von MD_MAPAL_PROFIL
"M_MAPAL_PROFIL_BIT_09"	M 2042.1	BOOL	// Angewähltes Profil der U-Achse Mapal: Bit von MD_MAPAL_PROFIL
"M_MAPAL_PROFIL_BIT_10"	M 2042.2	BOOL	// Angewähltes Profil der U-Achse Mapal: Bit von MD_MAPAL_PROFIL
"M_MAPAL_PROFIL_BIT_11"	M 2042.3	BOOL	// Angewähltes Profil der U-Achse Mapal: Bit von MD_MAPAL_PROFIL
"M_MAPAL_PROFIL_BIT_12"	M 2042.4	BOOL	// Angewähltes Profil der U-Achse Mapal: Bit von MD_MAPAL_PROFIL
"M_MAPAL_PROFIL_BIT_13"	M 2042.5	BOOL	// Angewähltes Profil der U-Achse Mapal: Bit von MD_MAPAL_PROFIL
"M_MAPAL_PROFIL_BIT_14"	M 2042.6	BOOL	// Angewähltes Profil der U-Achse Mapal: Bit von MD_MAPAL_PROFIL
"M_MAPAL_PROFIL_BIT_15"	M 2042.7	BOOL	// Angewähltes Profil der U-Achse Mapal: Bit von MD_MAPAL_PROFIL
"M_MAPAL_PROFIL_BIT_00"	M 2043.0	BOOL	// Angewähltes Profil der U-Achse Mapal: Bit von MD_MAPAL_PROFIL
"M_MAPAL_PROFIL_BIT_01"	M 2043.1	BOOL	// Angewähltes Profil der U-Achse Mapal: Bit von MD_MAPAL_PROFIL
"M_MAPAL_PROFIL_BIT_02"	M 2043.2	BOOL	// Angewähltes Profil der U-Achse Mapal: Bit von MD_MAPAL_PROFIL
"M_MAPAL_PROFIL_BIT_03"	M 2043.3	BOOL	// Angewähltes Profil der U-Achse Mapal: Bit von MD_MAPAL_PROFIL
"M_MAPAL_PROFIL_BIT_04"	M 2043.4	BOOL	// Angewähltes Profil der U-Achse Mapal: Bit von MD_MAPAL_PROFIL
"M_MAPAL_PROFIL_BIT_05"	M 2043.5	BOOL	// Angewähltes Profil der U-Achse Mapal: Bit von MD_MAPAL_PROFIL
"M_MAPAL_PROFIL_BIT_06"	M 2043.6	BOOL	// Angewähltes Profil der U-Achse Mapal: Bit von MD_MAPAL_PROFIL
"M_MAPAL_PROFIL_BIT_07"	M 2043.7	BOOL	// Angewähltes Profil der U-Achse Mapal: Bit von MD_MAPAL_PROFIL
"O_GEN_OPTWAVE_RD"	M 2061.0	BOOL	// M-AUSGANG: Signalband Farbe Rot
"O_GEN_OPTWAVE_GN"	M 2061.2	BOOL	// M-AUSGANG: Signalband Farbe Grün
"O_GEN_OPTWAVE_BU"	M 2061.3	BOOL	// M-AUSGANG: Signalband Farbe Blau
"M_PC_LIFT_MID_PERIPH_E"	M 2066.2	BOOL	// Schneller Eingang Palettenwechsler mitte E66.2 Peripherie-Eingang
"M_WZ_SPA_GEL_PERIPH_E"	M 2067.4	BOOL	// Schneller Eingang Werkzeugspanner gelöst E63.4 Peripherie-Eingang
"M_WZ_SPA_GES_PERIPH_E"	M 2067.5	BOOL	// Schneller Eingang Werkzeugspanner gespannt E63.5 Peripherie-Eingang
"M_WZ_SPA_GES_OW_PERIPH_E"	M 2067.7	BOOL	// Schneller Eingang Werkzeugspanner gespannt ohne Wz E63.7 Peripherie-Eingang
"M_PS_DRIVES_EN_PERIPH_E"	M 2068.7	BOOL	// Digitaleingabemodul , PROFIsafe V2 (E505.7 = DB_SPL".ISX_PS_DRIVES_EN_CNC)
"M_PC_LIFT_UP_PERIPH_A"	M 2076.0	BOOL	// Schneller Ausgang Palettenwechsler nach oben A76.0 Peripherie-Ausgang
"M_PC_LIFT_DOWN_PERIPH_A"	M 2076.1	BOOL	// Schneller Ausgang Palettenwechsler nach unten A76.1 Peripherie-Ausgang
"M_READY_WZ_MELDEN"	M 2435.7	BOOL
"M_FP_Reset_FMS_Prog_END"	M 2453.0	BOOL
"M_FP_Keine _Pal_vorhande"	M 2453.1	BOOL
"M_FP_FMS_WZ_BRUCH"	M 2453.2	BOOL
"MB_Systemtakt"	MB 1	BYTE
"MB_OB1_Zyklen"	MB 2	BYTE	// OB1 Zyklen
"MB_Takt"	MB 7	BYTE
"MB_Takt_Speicher"	MB 8	BYTE
"MB_Anlauf_Merker"	MB 9	BYTE	// Anlauf 1.bis 8.Zyklus bleibt anstehen
"MB_10s_Takt_Count"	MB 29	BYTE	// Merkerbyte 10 Sekunden Takt
"MW_BGH_Vorschub_LSB"	MB 41	BYTE	// niederwertiges Byte von MW_BHG_Vorschub
"MB_SKZ_WZB"	MB 54	BYTE	// Schrittkette WZ-Bruch
"MB_SKZ_WZB_Lesen"	MB 56	BYTE	// Schrittkette Lesen WZ-Bruch
"MB_SKZ_DrehDurch"	MB 61	BYTE	// Schrittkette Schmierung DrehDurchführung
"MB_Wert_0"	MB 66	BYTE
"MB_FD_Kuehl_Agg_Count"	MB 74	BYTE
"MB_Kuehl_Agg_Count"	MB 75	BYTE	// Counter Kühlaggregat
"MB_SZ_MAN_WZW"	MB 81	BYTE	// MAN WZW: Schrittkettenzaehler
"MB_Max_Paus_Dauer"	MB 86	BYTE	// GT MAG1:
"MB_Max_Pein_Dauer"	MB 87	BYTE	// GT MAG1:
"MB_Min_Paus_Dauer"	MB 88	BYTE	// GT MAG1:
"MB_Min_Pein_Dauer"	MB 89	BYTE	// GT MAG1:
"MB_Aus_Zaehler"	MB 90	BYTE	// GT MAG1: Auszeit Zaehler
"MB_Kal_Zaehler"	MB 91	BYTE	// GT MAG1: Kaliebrierungs Zaehler
"MB_Paus_Zaehler"	MB 93	BYTE	// GT MAG1: Puls Aus Zaehler
"MB_Pein_Zaehler"	MB 94	BYTE	// GT MAG1: Puls Ein Zaehler
"MB_SKZ_Abl_Mag1"	MB 95	BYTE	// GT MAG1: Schrittkettenzaehler Ablauf Magazin 1
"MB_SKZ_Kal_Mag1"	MB 96	BYTE	// GT MAG1: Schrittkettenzaehler Kalibrierung Magazin 1
"MB_SKZ_TOut_Mag1"	MB 97	BYTE	// GT MAG1: Schrittkettenzaehler Tout Magazin1
"MB_Mag_Fehler_Nr"	MB 98	BYTE	// GT MAG1:Fehler Nr von Ablaufmodul
"MB_Mag_Anforderung"	MB 106	BYTE	// Magazin Anforderung
"B_MA_SKZ_Oelstand"	MB 130	BYTE	// MA: Schrittkette Oelstand
"B_MA_SKZ_MaschineEin"	MB 131	BYTE	// MA: Schrittkette Maschine Ein
